KUKA KRL program: MyProgram_199().src

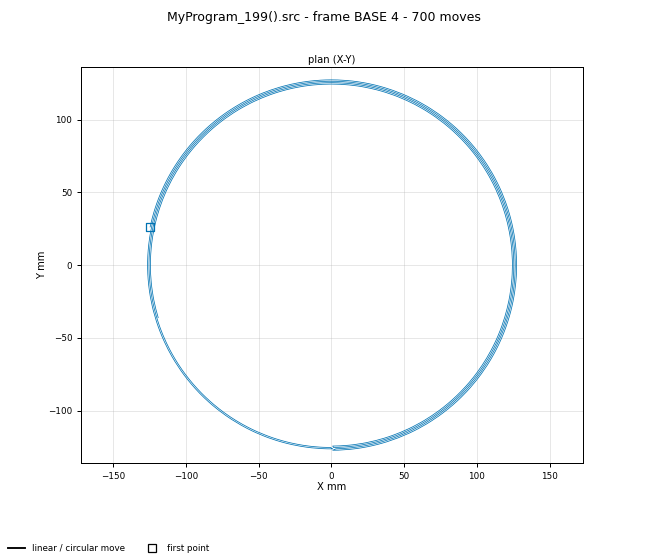
[picture p0: tool path of MyProgram_199().src in frame BASE 4, 700 of 700 moves have a stored position in this frame; points joined in program order, loops and branches not executed]
&ACCESS RVP
&REL 1
&PARAM TEMPLATE = C:\KRC\Roboter\Template\vorgabe
&PARAM EDITMASK = *
DEF MyProgram_199()
; ---- Setting reference (Base) ----
$BASE = BASE_DATA[4]

; --------------------------
; ---- Setting tool (TCP) ----
$TOOL = TOOL_DATA[3]
; --------------------------

$VEL.CP = VEL_APROX_PRINT
Startdeposition()
$VEL.CP = VEL_PRINT
LIN {X -124.5272,Y 26.175,Z 143,A 164.1665,B 24.1206,C -1.3898,E1 24.0018,E2 642.4936} C_DIS
LIN {X -123.2727,Y 31.5525,Z 143,A 161.827,B 24.1198,C -1.4042,E1 24.0033,E2 644.8119} C_DIS
LIN {X -122.0443,Y 36.0123,Z 143,A 159.352,B 24.1204,C -1.3939,E1 24.0052,E2 647.3273} C_DIS
LIN {X -120.9556,Y 39.5205,Z 143,A 158.1178,B 24.1191,C -1.4173,E1 24.0063,E2 648.5112} C_DIS
LIN {X -119.8977,Y 42.6203,Z 143,A 156.6922,B 24.1187,C -1.4241,E1 24.0075,E2 649.9285} C_DIS
LIN {X -118.7019,Y 45.8427,Z 143,A 154.9477,B 24.1189,C -1.4203,E1 24.0093,E2 651.6925} C_DIS
LIN {X -117.3172,Y 49.2782,Z 143,A 152.7105,B 24.12,C -1.4008,E1 24.0118,E2 653.9905} C_DIS
LIN {X -115.3752,Y 53.668,Z 143,A 151.1857,B 24.1181,C -1.435,E1 24.0135,E2 655.44} C_DIS
LIN {X -114.0458,Y 56.4373,Z 143,A 149.7836,B 24.1179,C -1.4383,E1 24.0152,E2 656.8417} C_DIS
LIN {X -112.4501,Y 59.5546,Z 143,A 147.9643,B 24.1183,C -1.4324,E1 24.0175,E2 658.6856} C_DIS
LIN {X -109.8769,Y 64.1814,Z 143,A 145.6973,B 24.1176,C -1.4445,E1 24.0207,E2 660.9353} C_DIS
LIN {X -107.6931,Y 67.7812,Z 143,A 143.7781,B 24.1173,C -1.4489,E1 24.0235,E2 662.8538} C_DIS
LIN {X -105.2252,Y 71.5528,Z 143,A 141.7365,B 24.1171,C -1.4541,E1 24.0266,E2 664.8932} C_DIS
LIN {X -102.675,Y 75.1662,Z 143,A 139.7684,B 24.1167,C -1.4606,E1 24.0298,E2 666.8553} C_DIS
LIN {X -100.2448,Y 78.3782,Z 143,A 137.8484,B 24.1167,C -1.4608,E1 24.0331,E2 668.7842} C_DIS
LIN {X -97.0311,Y 82.3229,Z 143,A 135.7966,B 24.1157,C -1.4774,E1 24.0367,E2 670.8052} C_DIS
LIN {X -94.8087,Y 84.8728,Z 143,A 133.5905,B 24.1172,C -1.4513,E1 24.0409,E2 673.0856} C_DIS
LIN {X -91.6928,Y 88.2304,Z 143,A 131.505,B 24.117,C -1.4554,E1 24.045,E2 675.1704} C_DIS
LIN {X -88.4466,Y 91.4838,Z 143,A 130.1435,B 24.1149,C -1.4916,E1 24.0475,E2 676.449} C_DIS
LIN {X -85.9693,Y 93.8157,Z 143,A 127.9481,B 24.1164,C -1.4659,E1 24.0522,E2 678.7167} C_DIS
LIN {X -82.7807,Y 96.64,Z 143,A 126.4601,B 24.115,C -1.4892,E1 24.0552,E2 680.1535} C_DIS
LIN {X -79.8951,Y 99.0396,Z 143,A 124.7629,B 24.1148,C -1.4926,E1 24.0589,E2 681.849} C_DIS
LIN {X -76.5158,Y 101.6731,Z 143,A 122.8099,B 24.1147,C -1.4957,E1 24.0632,E2 683.8019} C_DIS
LIN {X -72.9495,Y 104.2619,Z 143,A 120.7574,B 24.1147,C -1.4967,E1 24.0679,E2 685.8592} C_DIS
LIN {X -70.0309,Y 106.2438,Z 143,A 119.2441,B 24.1142,C -1.5032,E1 24.0714,E2 687.3619} C_DIS
LIN {X -66.2642,Y 108.6335,Z 143,A 116.7258,B 24.1153,C -1.4842,E1 24.0775,E2 689.9348} C_DIS
LIN {X -62.3439,Y 110.9293,Z 143,A 115.1658,B 24.1139,C -1.5095,E1 24.0811,E2 691.4375} C_DIS
LIN {X -58.8236,Y 112.834,Z 143,A 113.4971,B 24.1133,C -1.5186,E1 24.0852,E2 693.0888} C_DIS
LIN {X -56.2226,Y 114.1518,Z 143,A 112.1566,B 24.1133,C -1.5195,E1 24.0886,E2 694.4308} C_DIS
LIN {X -53.1753,Y 115.603,Z 143,A 110.5764,B 24.1133,C -1.5191,E1 24.0926,E2 696.016} C_DIS
LIN {X -50.3374,Y 116.8665,Z 143,A 109.2109,B 24.1131,C -1.5227,E1 24.096,E2 697.3761} C_DIS
LIN {X -47.1249,Y 118.1994,Z 143,A 106.7623,B 24.1153,C -1.4852,E1 24.1027,E2 699.9222} C_DIS
LIN {X -41.565,Y 120.2663,Z 143,A 104.0516,B 24.1152,C -1.4868,E1 24.1098,E2 702.6346} C_DIS
LIN {X -35.7294,Y 122.1272,Z 143,A 102.2253,B 24.1125,C -1.5319,E1 24.1144,E2 704.3534} C_DIS
LIN {X -32.6041,Y 122.9986,Z 143,A 100.6987,B 24.1126,C -1.5304,E1 24.1185,E2 705.8861} C_DIS
LIN {X -27.5686,Y 124.2263,Z 143,A 98.4289,B 24.1123,C -1.5355,E1 24.1247,E2 708.1466} C_DIS
LIN {X -23.6156,Y 125.0362,Z 143,A 96.5708,B 24.1123,C -1.5351,E1 24.1298,E2 710.0079} C_DIS
LIN {X -19.7127,Y 125.7106,Z 143,A 94.7472,B 24.1123,C -1.5346,E1 24.1348,E2 711.8346} C_DIS
LIN {X -16.2002,Y 126.2116,Z 143,A 93.0887,B 24.1125,C -1.5327,E1 24.1394,E2 713.4988} C_DIS
LIN {X -12.0343,Y 126.6763,Z 143,A 91.2754,B 24.1122,C -1.5372,E1 24.1444,E2 715.3025} C_DIS
LIN {X -7.2561,Y 127.0405,Z 143,A 88.7598,B 24.1131,C -1.5215,E1 24.1515,E2 717.8573} C_DIS
LIN {X -3.7963,Y 127.1904,Z 143,A 87.5723,B 24.1121,C -1.5392,E1 24.1547,E2 719.0017} C_DIS
LIN {X -0.1288,Y 127.248,Z 143,A 85.3654,B 24.1136,C -1.5137,E1 24.1611,E2 721.2708} C_DIS
LIN {X 4.2966,Y 127.1759,Z 143,A 83.9944,B 24.1119,C -1.5428,E1 24.1647,E2 722.5704} C_DIS
LIN {X 7.6952,Y 127.0138,Z 143,A 82.4885,B 24.1118,C -1.5441,E1 24.1689,E2 724.0726} C_DIS
LIN {X 10.3341,Y 126.8269,Z 143,A 81.1022,B 24.1123,C -1.5349,E1 24.1728,E2 725.4807} C_DIS
LIN {X 14.3391,Y 126.4382,Z 143,A 79.2362,B 24.1125,C -1.532,E1 24.178,E2 727.3524} C_DIS
LIN {X 18.3253,Y 125.9205,Z 143,A 77.4824,B 24.1124,C -1.5342,E1 24.1828,E2 729.0993} C_DIS
LIN {X 22.3665,Y 125.2654,Z 143,A 75.7321,B 24.1122,C -1.5379,E1 24.1876,E2 730.8386} C_DIS
LIN {X 25.9022,Y 124.5834,Z 143,A 73.9894,B 24.1126,C -1.5314,E1 24.1924,E2 732.595} C_DIS
LIN {X 29.705,Y 123.7307,Z 143,A 72.3528,B 24.1123,C -1.5361,E1 24.1969,E2 734.2179} C_DIS
LIN {X 32.889,Y 122.9226,Z 143,A 70.8777,B 24.1123,C -1.5353,E1 24.2008,E2 735.6924} C_DIS
LIN {X 36.7581,Y 121.8225,Z 143,A 68.3038,B 24.1145,C -1.4979,E1 24.208,E2 738.3531} C_DIS
LIN {X 41.983,Y 120.1214,Z 143,A 66.8144,B 24.1119,C -1.5425,E1 24.2116,E2 739.7305} C_DIS
LIN {X 48.6266,Y 117.5894,Z 143,A 63.5741,B 24.1122,C -1.5374,E1 24.2201,E2 742.976} C_DIS
LIN {X 52.3171,Y 115.9943,Z 143,A 61.5114,B 24.113,C -1.5232,E1 24.2254,E2 745.0681} C_DIS
LIN {X 57.8621,Y 113.3296,Z 143,A 58.8534,B 24.113,C -1.5251,E1 24.2321,E2 747.7141} C_DIS
LIN {X 60.9839,Y 111.6828,Z 143,A 57.1789,B 24.1133,C -1.5187,E1 24.2362,E2 749.3991} C_DIS
LIN {X 65.2332,Y 109.2553,Z 143,A 55.1366,B 24.113,C -1.5233,E1 24.2411,E2 751.4238} C_DIS
LIN {X 68.3421,Y 107.3384,Z 143,A 53.2984,B 24.1137,C -1.5113,E1 24.2455,E2 753.2852} C_DIS
LIN {X 73.4348,Y 103.9202,Z 143,A 50.8446,B 24.1131,C -1.5217,E1 24.2511,E2 755.7051} C_DIS
LIN {X 75.7493,Y 102.2458,Z 143,A 49.305,B 24.114,C -1.507,E1 24.2546,E2 757.2748} C_DIS
LIN {X 79.2546,Y 99.5529,Z 143,A 47.3269,B 24.1142,C -1.5039,E1 24.259,E2 759.2528} C_DIS
LIN {X 82.6863,Y 96.7222,Z 143,A 45.3026,B 24.1145,C -1.499,E1 24.2633,E2 761.281} C_DIS
LIN {X 85.935,Y 93.8473,Z 143,A 43.3542,B 24.1147,C -1.4953,E1 24.2673,E2 763.2304} C_DIS
LIN {X 89.2409,Y 90.7093,Z 143,A 41.3376,B 24.1148,C -1.4926,E1 24.2714,E2 765.2447} C_DIS
LIN {X 92.2645,Y 87.6327,Z 143,A 39.4106,B 24.115,C -1.4891,E1 24.2751,E2 767.1717} C_DIS
LIN {X 95.0993,Y 84.5477,Z 143,A 37.4842,B 24.1154,C -1.4828,E1 24.2788,E2 769.1045} C_DIS
LIN {X 98.0466,Y 81.1107,Z 143,A 35.1728,B 24.1165,C -1.4645,E1 24.283,E2 771.4495} C_DIS
LIN {X 100.4117,Y 78.1641,Z 143,A 34.1152,B 24.1149,C -1.4922,E1 24.2847,E2 772.4343} C_DIS
LIN {X 102.2377,Y 75.7602,Z 143,A 32.4351,B 24.116,C -1.4729,E1 24.2875,E2 774.1532} C_DIS
LIN {X 104.9494,Y 71.9562,Z 143,A 30.3694,B 24.1162,C -1.4694,E1 24.2909,E2 776.217} C_DIS
LIN {X 107.1146,Y 68.6917,Z 143,A 28.6075,B 24.1164,C -1.4649,E1 24.2935,E2 777.9808} C_DIS
LIN {X 110.4405,Y 63.2061,Z 143,A 26.0074,B 24.1161,C -1.4715,E1 24.2972,E2 780.5509} C_DIS
LIN {X 111.9201,Y 60.5483,Z 143,A 24.3472,B 24.1171,C -1.4531,E1 24.2995,E2 782.2467} C_DIS
LIN {X 114.1794,Y 56.1666,Z 143,A 22.2677,B 24.1171,C -1.4539,E1 24.3021,E2 784.3128} C_DIS
LIN {X 115.6591,Y 53.0539,Z 143,A 20.7526,B 24.1172,C -1.4513,E1 24.3039,E2 785.8258} C_DIS
LIN {X 116.9946,Y 50.0412,Z 143,A 18.1864,B 24.1204,C -1.393,E1 24.3069,E2 788.5191} C_DIS
LIN {X 119.5516,Y 43.5801,Z 143,A 15.4723,B 24.1198,C -1.4042,E1 24.3094,E2 791.1903} C_DIS
LIN {X 121.1576,Y 38.8909,Z 143,A 13.3661,B 24.1198,C -1.4037,E1 24.3112,E2 793.2853} C_DIS
LIN {X 122.4466,Y 34.6207,Z 143,A 12.1149,B 24.1181,C -1.4356,E1 24.3121,E2 794.4515} C_DIS
LIN {X 123.2167,Y 31.773,Z 143,A 10.5319,B 24.119,C -1.4186,E1 24.3133,E2 796.0665} C_DIS
LIN {X 124.0498,Y 28.3427,Z 143,A 8.9948,B 24.1192,C -1.4162,E1 24.3143,E2 797.6} C_DIS
LIN {X 124.7446,Y 25.1102,Z 143,A 7.5368,B 24.1193,C -1.4131,E1 24.3151,E2 799.0569} C_DIS
LIN {X 125.4856,Y 21.0966,Z 143,A 5.7162,B 24.1196,C -1.4081,E1 24.316,E2 800.8785} C_DIS
LIN {X 126.0104,Y 17.6965,Z 143,A 4.0643,B 24.1202,C -1.398,E1 24.3167,E2 802.5449} C_DIS
LIN {X 126.5349,Y 13.4408,Z 143,A 2.2564,B 24.1202,C -1.398,E1 24.3172,E2 804.3417} C_DIS
LIN {X 126.8936,Y 9.475,Z 143,A 0.4251,B 24.1206,C -1.3902,E1 24.3177,E2 806.1805} C_DIS
LIN {X 127.2222,Y 2.5341,Z 143,A -2.4521,B 24.1205,C -1.3928,E1 24.318,E2 809.0338} C_DIS
LIN {X 127.1851,Y -3.9522,Z 143,A -5.6524,B 24.1217,C -1.369,E1 24.318,E2 812.272} C_DIS
LIN {X 127.0034,Y -7.8649,Z 143,A -7.2947,B 24.1217,C -1.3694,E1 24.3177,E2 813.9033} C_DIS
LIN {X 126.673,Y -12.0688,Z 143,A -9.1796,B 24.122,C -1.3639,E1 24.3172,E2 815.79} C_DIS
LIN {X 125.9979,Y -17.7836,Z 143,A -11.5619,B 24.1219,C -1.366,E1 24.3164,E2 818.1524} C_DIS
LIN {X 125.5414,Y -20.7622,Z 143,A -13.1259,B 24.1227,C -1.3511,E1 24.3157,E2 819.7433} C_DIS
LIN {X 124.8202,Y -24.7388,Z 143,A -15.3256,B 24.124,C -1.3259,E1 24.3145,E2 821.9908} C_DIS
LIN {X 124.0308,Y -28.4258,Z 143,A -16.5022,B 24.1229,C -1.3468,E1 24.3138,E2 823.1094} C_DIS
LIN {X 123.3013,Y -31.4399,Z 143,A -17.9511,B 24.1233,C -1.3397,E1 24.3128,E2 824.5671} C_DIS
LIN {X 122.3396,Y -35.0032,Z 143,A -20.1035,B 24.1248,C -1.3095,E1 24.3112,E2 826.78} C_DIS
LIN {X 121.1722,Y -38.8452,Z 143,A -21.418,B 24.1239,C -1.3287,E1 24.3101,E2 828.0401} C_DIS
LIN {X 119.4922,Y -43.745,Z 143,A -23.6832,B 24.1241,C -1.3247,E1 24.308,E2 830.3016} C_DIS
LIN {X 118.3727,Y -46.6894,Z 143,A -25.5245,B 24.1254,C -1.2989,E1 24.3061,E2 832.1951} C_DIS
LIN {X 117.0359,Y -49.9411,Z 143,A -27.4139,B 24.1264,C -1.2787,E1 24.304,E2 834.1231} C_DIS
LIN {X 114.8725,Y -54.735,Z 143,A -28.7689,B 24.1242,C -1.3226,E1 24.3025,E2 835.3636} C_DIS
LIN {X 113.2953,Y -57.9294,Z 143,A -30.6449,B 24.1251,C -1.3039,E1 24.3001,E2 837.2746} C_DIS
LIN {X 111.5668,Y -61.1965,Z 143,A -32.3955,B 24.1256,C -1.2945,E1 24.2978,E2 839.0385} C_DIS
LIN {X 109.5112,Y -64.8038,Z 143,A -34.2914,B 24.1259,C -1.2877,E1 24.2951,E2 840.9408} C_DIS
LIN {X 106.9666,Y -68.9229,Z 143,A -37.4263,B 24.1286,C -1.2337,E1 24.2902,E2 844.1907} C_DIS
LIN {X 102.9212,Y -74.8288,Z 143,A -39.4667,B 24.1261,C -1.2838,E1 24.2871,E2 846.0989} C_DIS
LIN {X 99.7193,Y -79.045,Z 143,A -42.1819,B 24.1273,C -1.2607,E1 24.2824,E2 848.8571} C_DIS
LIN {X 95.2135,Y -84.4186,Z 143,A -44.9279,B 24.1267,C -1.273,E1 24.2775,E2 851.56} C_DIS
LIN {X 92.859,Y -87.0024,Z 143,A -46.6893,B 24.1273,C -1.2596,E1 24.2741,E2 853.346} C_DIS
LIN {X 88.9185,Y -91.0254,Z 143,A -49.4625,B 24.1282,C -1.2415,E1 24.2686,E2 856.1511} C_DIS
LIN {X 86.4722,Y -93.3528,Z 143,A -50.6453,B 24.1276,C -1.2547,E1 24.2663,E2 857.2968} C_DIS
LIN {X 83.4676,Y -96.0484,Z 143,A -52.5339,B 24.128,C -1.2469,E1 24.2623,E2 859.1965} C_DIS
LIN {X 79.6258,Y -99.2568,Z 143,A -55.2366,B 24.1293,C -1.2196,E1 24.2563,E2 861.9551} C_DIS
LIN {X 76.152,Y -101.946,Z 143,A -56.4363,B 24.1276,C -1.254,E1 24.2539,E2 863.0665} C_DIS
LIN {X 73.7292,Y -103.7121,Z 143,A -58.3085,B 24.129,C -1.2252,E1 24.2495,E2 865.0021} C_DIS
LIN {X 68.4798,Y -107.2502,Z 143,A -60.5853,B 24.1279,C -1.248,E1 24.2443,E2 867.2154} C_DIS
LIN {X 65.0588,Y -109.3592,Z 143,A -62.7183,B 24.1289,C -1.2285,E1 24.2391,E2 869.3889} C_DIS
LIN {X 59.4478,Y -112.5062,Z 143,A -65.3808,B 24.1285,C -1.2349,E1 24.2327,E2 872.0277} C_DIS
LIN {X 57.032,Y -113.7522,Z 143,A -66.8895,B 24.1293,C -1.2188,E1 24.2288,E2 873.5714} C_DIS
LIN {X 53.4352,Y -115.4828,Z 143,A -68.5743,B 24.1292,C -1.2215,E1 24.2246,E2 875.2452} C_DIS
LIN {X 45.816,Y -118.7123,Z 143,A -71.9325,B 24.1286,C -1.2341,E1 24.2161,E2 878.5644} C_DIS
LIN {X 38.1325,Y -121.3998,Z 143,A -75.7888,B 24.1293,C -1.2198,E1 24.2059,E2 882.4475} C_DIS
LIN {X 34.5937,Y -122.4542,Z 143,A -77.3703,B 24.1292,C -1.2219,E1 24.2016,E2 884.021} C_DIS
LIN {X 31.4599,Y -123.2962,Z 143,A -79.0235,B 24.1297,C -1.211,E1 24.1971,E2 885.6982} C_DIS
LIN {X 28.2059,Y -124.081,Z 143,A -80.5262,B 24.1297,C -1.2098,E1 24.193,E2 887.2017} C_DIS
LIN {X 24.8866,Y -124.7901,Z 143,A -82.181,B 24.1301,C -1.2023,E1 24.1884,E2 888.8727} C_DIS
LIN {X 20.9689,Y -125.5069,Z 143,A -83.8399,B 24.1299,C -1.2074,E1 24.1839,E2 890.5173} C_DIS
LIN {X 17.5219,Y -126.0353,Z 143,A -85.6002,B 24.1303,C -1.1971,E1 24.179,E2 892.3011} C_DIS
LIN {X 12.5269,Y -126.6291,Z 143,A -87.4842,B 24.1295,C -1.2142,E1 24.1739,E2 894.142} C_DIS
LIN {X 4.6976,Y -127.1602,Z 143,A -91.0863,B 24.1298,C -1.2093,E1 24.1638,E2 897.7545} C_DIS
LIN {X 0.9052,Y -127.2215,Z 143,A -92.4328,B 24.1289,C -1.2265,E1 24.1602,E2 899.0586} C_DIS
Enddeposition()
LIN {X 0.9052,Y -127.2215,Z 143,A -92.4328,B 24.1289,C -1.2265,E1 24.1602,E2 899.0586} C_DIS
Startdeposition()
$VEL.CP = VEL_PRINT
LIN {X 3.0703,Y -126.2444,Z 143,A -90.8348,B 23.3783,C -1.1238,E1 23.4098,E2 897.6156} C_DIS
LIN {X 9.0133,Y -125.959,Z 143,A -88.2436,B 23.3785,C -1.1199,E1 23.4169,E2 895.0355} C_DIS
LIN {X 12.8377,Y -125.6284,Z 143,A -86.5864,B 23.3786,C -1.1168,E1 23.4215,E2 893.3871} C_DIS
LIN {X 17.843,Y -125.0139,Z 143,A -84.275,B 23.3786,C -1.1194,E1 23.4279,E2 891.0714} C_DIS
LIN {X 21.7376,Y -124.3968,Z 143,A -82.4343,B 23.3784,C -1.1231,E1 23.433,E2 889.2232} C_DIS
LIN {X 25.0313,Y -123.7751,Z 143,A -80.9906,B 23.3784,C -1.1208,E1 23.437,E2 887.7872} C_DIS
LIN {X 28.5169,Y -123.0193,Z 143,A -79.268,B 23.3782,C -1.1272,E1 23.4417,E2 886.051} C_DIS
LIN {X 32.3455,Y -122.068,Z 143,A -77.6252,B 23.3784,C -1.1221,E1 23.4461,E2 884.4238} C_DIS
LIN {X 35.6782,Y -121.1359,Z 143,A -75.87,B 23.3779,C -1.1326,E1 23.4509,E2 882.6453} C_DIS
LIN {X 42.4632,Y -118.9277,Z 143,A -72.6202,B 23.3777,C -1.1372,E1 23.4595,E2 879.3908} C_DIS
LIN {X 46.97,Y -117.2205,Z 143,A -70.8654,B 23.3785,C -1.1196,E1 23.4639,E2 877.6844} C_DIS
LIN {X 52.3569,Y -114.9174,Z 143,A -67.8848,B 23.3776,C -1.1389,E1 23.4717,E2 874.6631} C_DIS
LIN {X 55.7551,Y -113.3055,Z 143,A -66.2507,B 23.3776,C -1.1382,E1 23.4757,E2 873.0354} C_DIS
LIN {X 61.2211,Y -110.45,Z 143,A -63.4821,B 23.3776,C -1.1415,E1 23.4826,E2 870.2669} C_DIS
LIN {X 64.3168,Y -108.6772,Z 143,A -61.8595,B 23.3774,C -1.1446,E1 23.4865,E2 868.6418} C_DIS
LIN {X 67.2956,Y -106.8576,Z 143,A -60.2613,B 23.3772,C -1.1483,E1 23.4903,E2 867.0397} C_DIS
LIN {X 69.4871,Y -105.4456,Z 143,A -59.0358,B 23.377,C -1.1527,E1 23.4932,E2 865.8076} C_DIS
LIN {X 74.8729,Y -101.6922,Z 143,A -56.0676,B 23.3767,C -1.1583,E1 23.4999,E2 862.8364} C_DIS
LIN {X 78.5319,Y -98.8938,Z 143,A -53.9887,B 23.3766,C -1.1623,E1 23.5045,E2 860.7558} C_DIS
LIN {X 83.5514,Y -94.6911,Z 143,A -51.0321,B 23.3763,C -1.1683,E1 23.5108,E2 857.7965} C_DIS
LIN {X 88.903,Y -89.6855,Z 143,A -47.0482,B 23.3743,C -1.2087,E1 23.519,E2 853.7291} C_DIS
LIN {X 92.7346,Y -85.7184,Z 143,A -45.2748,B 23.3758,C -1.179,E1 23.5222,E2 852.0384} C_DIS
LIN {X 97.8322,Y -79.8504,Z 143,A -40.9889,B 23.3735,C -1.2257,E1 23.5301,E2 847.6566} C_DIS
LIN {X 101.4084,Y -75.257,Z 143,A -39.1077,B 23.375,C -1.1953,E1 23.5331,E2 845.8614} C_DIS
LIN {X 103.0955,Y -72.9286,Z 143,A -36.7932,B 23.3723,C -1.249,E1 23.537,E2 843.4244} C_DIS
LIN {X 107.074,Y -66.9512,Z 143,A -34.5488,B 23.3744,C -1.2078,E1 23.5402,E2 841.2955} C_DIS
LIN {X 109.3173,Y -63.2216,Z 143,A -32.6201,B 23.3742,C -1.2113,E1 23.5429,E2 839.3688} C_DIS
LIN {X 111.3593,Y -59.5517,Z 143,A -30.6871,B 23.3739,C -1.2182,E1 23.5455,E2 837.4292} C_DIS
LIN {X 113.161,Y -56.048,Z 143,A -29.16,B 23.3742,C -1.2108,E1 23.5474,E2 835.9295} C_DIS
LIN {X 116.3932,Y -48.9847,Z 143,A -25.5078,B 23.3734,C -1.2277,E1 23.5516,E2 832.2563} C_DIS
LIN {X 117.5948,Y -46.0252,Z 143,A -24.1792,B 23.3734,C -1.2262,E1 23.553,E2 830.9393} C_DIS
LIN {X 118.592,Y -43.3943,Z 143,A -22.4227,B 23.3721,C -1.2539,E1 23.5547,E2 829.1239} C_DIS
LIN {X 119.7735,Y -40.0138,Z 143,A -21.3647,B 23.3732,C -1.231,E1 23.5556,E2 828.13} C_DIS
LIN {X 121.5558,Y -34.2204,Z 143,A -18.5087,B 23.3725,C -1.2448,E1 23.5579,E2 825.2567} C_DIS
LIN {X 122.3741,Y -31.1673,Z 143,A -17.1035,B 23.3724,C -1.248,E1 23.5589,E2 823.8523} C_DIS
LIN {X 123.4702,Y -26.4942,Z 143,A -14.8735,B 23.3719,C -1.2575,E1 23.5603,E2 821.6123} C_DIS
LIN {X 124.2579,Y -22.5139,Z 143,A -13.0509,B 23.3716,C -1.2625,E1 23.5613,E2 819.7887} C_DIS
LIN {X 124.864,Y -18.8685,Z 143,A -10.8775,B 23.3701,C -1.2926,E1 23.5622,E2 817.5537} C_DIS
LIN {X 125.4288,Y -14.6483,Z 143,A -9.4064,B 23.371,C -1.276,E1 23.5627,E2 816.1336} C_DIS
LIN {X 125.8412,Y -10.5292,Z 143,A -7.6065,B 23.3708,C -1.2782,E1 23.5631,E2 814.3396} C_DIS
LIN {X 126.0963,Y -6.8457,Z 143,A -6.0912,B 23.371,C -1.2757,E1 23.5634,E2 812.8403} C_DIS
LIN {X 126.2797,Y -0.8325,Z 143,A -3.6263,B 23.3712,C -1.2715,E1 23.5636,E2 810.4018} C_DIS
LIN {X 126.2604,Y 2.2898,Z 143,A -1.8926,B 23.3701,C -1.2917,E1 23.5636,E2 808.6286} C_DIS
LIN {X 126.0769,Y 7.1985,Z 143,A 0.3117,B 23.3698,C -1.2976,E1 23.5633,E2 806.4235} C_DIS
LIN {X 125.8526,Y 10.3945,Z 143,A 1.8479,B 23.3694,C -1.3064,E1 23.563,E2 804.8751} C_DIS
LIN {X 125.4982,Y 14.048,Z 143,A 3.5727,B 23.3689,C -1.3146,E1 23.5624,E2 803.1407} C_DIS
LIN {X 125.0207,Y 17.7952,Z 143,A 5.1722,B 23.3689,C -1.3145,E1 23.5619,E2 801.5518} C_DIS
LIN {X 124.4344,Y 21.5277,Z 143,A 6.8886,B 23.3686,C -1.32,E1 23.5611,E2 799.8324} C_DIS
LIN {X 123.7908,Y 24.954,Z 143,A 8.4425,B 23.3685,C -1.3236,E1 23.5602,E2 798.2792} C_DIS
LIN {X 123.0633,Y 28.3247,Z 143,A 10.0144,B 23.3682,C -1.3288,E1 23.5593,E2 796.704} C_DIS
LIN {X 122.0814,Y 32.2955,Z 143,A 11.7987,B 23.3681,C -1.331,E1 23.5581,E2 794.9253} C_DIS
LIN {X 121.1474,Y 35.6388,Z 143,A 14.0642,B 23.3659,C -1.37,E1 23.5562,E2 792.5762} C_DIS
LIN {X 119.6438,Y 40.4033,Z 143,A 15.7815,B 23.3671,C -1.3496,E1 23.5548,E2 790.9204} C_DIS
LIN {X 118.3757,Y 43.9782,Z 143,A 17.2604,B 23.3674,C -1.3429,E1 23.5534,E2 789.4673} C_DIS
LIN {X 116.1309,Y 49.6053,Z 143,A 20.1647,B 23.3666,C -1.3585,E1 23.5503,E2 786.5411} C_DIS
LIN {X 114.8576,Y 52.4863,Z 143,A 21.6205,B 23.3663,C -1.3639,E1 23.5486,E2 785.0803} C_DIS
LIN {X 112.9208,Y 56.5349,Z 143,A 23.7059,B 23.3658,C -1.372,E1 23.546,E2 782.9865} C_DIS
LIN {X 110.8846,Y 60.4304,Z 143,A 25.2832,B 23.3666,C -1.3572,E1 23.544,E2 781.4553} C_DIS
LIN {X 109.4448,Y 62.9996,Z 143,A 27.2771,B 23.3647,C -1.3929,E1 23.5412,E2 779.3829} C_DIS
LIN {X 107.4784,Y 66.3002,Z 143,A 28.669,B 23.3654,C -1.3804,E1 23.5392,E2 778.0301} C_DIS
LIN {X 105.2267,Y 69.819,Z 143,A 30.5814,B 23.365,C -1.3861,E1 23.5363,E2 776.1136} C_DIS
LIN {X 102.9014,Y 73.2022,Z 143,A 32.4389,B 23.3648,C -1.3906,E1 23.5333,E2 774.2546} C_DIS
LIN {X 100.3238,Y 76.6966,Z 143,A 34.5444,B 23.3641,C -1.4021,E1 23.5297,E2 772.1312} C_DIS
LIN {X 96.7287,Y 81.1836,Z 143,A 36.9626,B 23.3643,C -1.3991,E1 23.5255,E2 769.7326} C_DIS
LIN {X 93.8377,Y 84.5094,Z 143,A 38.9811,B 23.364,C -1.4046,E1 23.5217,E2 767.7101} C_DIS
LIN {X 90.8868,Y 87.6748,Z 143,A 40.9026,B 23.3639,C -1.4069,E1 23.518,E2 765.7917} C_DIS
LIN {X 87.9767,Y 90.5945,Z 143,A 42.7877,B 23.3636,C -1.4116,E1 23.5143,E2 763.9033} C_DIS
LIN {X 84.6059,Y 93.7506,Z 143,A 44.8759,B 23.3634,C -1.4156,E1 23.51,E2 761.8142} C_DIS
LIN {X 81.3687,Y 96.5734,Z 143,A 46.8072,B 23.3632,C -1.4186,E1 23.5059,E2 759.8836} C_DIS
LIN {X 78.0166,Y 99.3007,Z 143,A 48.5897,B 23.3635,C -1.4138,E1 23.502,E2 758.1204} C_DIS
LIN {X 75.0876,Y 101.5344,Z 143,A 50.2862,B 23.3632,C -1.418,E1 23.4983,E2 756.4199} C_DIS
LIN {X 71.4837,Y 104.1022,Z 143,A 52.5264,B 23.3624,C -1.4324,E1 23.4931,E2 754.1517} C_DIS
LIN {X 67.4019,Y 106.7905,Z 143,A 54.5602,B 23.3627,C -1.4273,E1 23.4883,E2 752.138} C_DIS
LIN {X 64.1824,Y 108.7562,Z 143,A 56.0506,B 23.3631,C -1.4194,E1 23.4848,E2 750.6723} C_DIS
LIN {X 61.8868,Y 110.0784,Z 143,A 57.5822,B 23.3621,C -1.4367,E1 23.481,E2 749.1022} C_DIS
LIN {X 58.555,Y 111.8843,Z 143,A 59.2144,B 23.3622,C -1.4349,E1 23.477,E2 747.4794} C_DIS
LIN {X 53.7161,Y 114.2889,Z 143,A 61.7393,B 23.3619,C -1.4414,E1 23.4707,E2 744.9454} C_DIS
LIN {X 50.168,Y 115.8876,Z 143,A 63.373,B 23.3621,C -1.4373,E1 23.4665,E2 743.3265} C_DIS
LIN {X 46.8946,Y 117.2509,Z 143,A 65.5891,B 23.3603,C -1.4674,E1 23.4606,E2 741.0399} C_DIS
LIN {X 42.404,Y 118.9491,Z 143,A 67.248,B 23.3617,C -1.4451,E1 23.4564,E2 739.4409} C_DIS
LIN {X 39.0441,Y 120.0948,Z 143,A 69.1038,B 23.3609,C -1.4578,E1 23.4514,E2 737.5567} C_DIS
LIN {X 35.8172,Y 121.0952,Z 143,A 70.2942,B 23.3618,C -1.4431,E1 23.4483,E2 736.4058} C_DIS
LIN {X 32.6406,Y 121.9893,Z 143,A 71.7276,B 23.3618,C -1.4411,E1 23.4445,E2 734.9798} C_DIS
LIN {X 29.5465,Y 122.7754,Z 143,A 73.2271,B 23.3618,C -1.4444,E1 23.4404,E2 733.4745} C_DIS
LIN {X 25.6496,Y 123.6493,Z 143,A 75.0835,B 23.3615,C -1.4473,E1 23.4353,E2 731.6132} C_DIS
LIN {X 21.7187,Y 124.4002,Z 143,A 76.8644,B 23.3615,C -1.4464,E1 23.4304,E2 729.8367} C_DIS
LIN {X 17.8497,Y 125.0129,Z 143,A 78.6606,B 23.3615,C -1.4479,E1 23.4255,E2 728.0388} C_DIS
LIN {X 13.7932,Y 125.5256,Z 143,A 80.4772,B 23.3615,C -1.4465,E1 23.4204,E2 726.2271} C_DIS
LIN {X 10.3945,Y 125.8526,Z 143,A 82.0898,B 23.3614,C -1.4495,E1 23.4159,E2 724.6078} C_DIS
LIN {X 7.597,Y 126.0523,Z 143,A 83.4759,B 23.3611,C -1.4547,E1 23.412,E2 723.2092} C_DIS
LIN {X 3.3796,Y 126.2358,Z 143,A 85.4736,B 23.3609,C -1.4583,E1 23.4064,E2 721.2029} C_DIS
LIN {X -1.4286,Y 126.2747,Z 143,A 87.4404,B 23.3615,C -1.4481,E1 23.401,E2 719.2619} C_DIS
LIN {X -4.5585,Y 126.1992,Z 143,A 88.7783,B 23.3617,C -1.444,E1 23.3973,E2 717.9342} C_DIS
LIN {X -10.2698,Y 125.8631,Z 143,A 91.4685,B 23.3615,C -1.4472,E1 23.3898,E2 715.2348} C_DIS
LIN {X -13.8004,Y 125.5248,Z 143,A 93.0275,B 23.3617,C -1.4442,E1 23.3855,E2 713.6827} C_DIS
LIN {X -17.827,Y 125.0162,Z 143,A 94.8643,B 23.3617,C -1.4428,E1 23.3804,E2 711.8477} C_DIS
LIN {X -21.5271,Y 124.4345,Z 143,A 96.6906,B 23.3615,C -1.4473,E1 23.3753,E2 710.0084} C_DIS
LIN {X -25.061,Y 123.7691,Z 143,A 98.1808,B 23.362,C -1.4397,E1 23.3713,E2 708.5355} C_DIS
LIN {X -28.2376,Y 123.0832,Z 143,A 99.7743,B 23.3617,C -1.4437,E1 23.3669,E2 706.9297} C_DIS
LIN {X -33.339,Y 121.8023,Z 143,A 102.1269,B 23.362,C -1.4398,E1 23.3606,E2 704.5832} C_DIS
LIN {X -37.8031,Y 120.4897,Z 143,A 104.6963,B 23.3609,C -1.4578,E1 23.3536,E2 701.9634} C_DIS
LIN {X -41.8081,Y 119.1599,Z 143,A 105.9845,B 23.3627,C -1.4277,E1 23.3504,E2 700.7487} C_DIS
LIN {X -46.4132,Y 117.4439,Z 143,A 108.3333,B 23.3625,C -1.43,E1 23.3442,E2 698.3889} C_DIS
LIN {X -49.7738,Y 116.058,Z 143,A 109.9891,B 23.3627,C -1.4279,E1 23.34,E2 696.7341} C_DIS
LIN {X -52.7954,Y 114.7147,Z 143,A 111.5069,B 23.3627,C -1.4265,E1 23.3361,E2 695.2161} C_DIS
LIN {X -55.7129,Y 113.3263,Z 143,A 112.9483,B 23.3629,C -1.4231,E1 23.3325,E2 693.7792} C_DIS
LIN {X -58.5976,Y 111.8619,Z 143,A 114.4346,B 23.363,C -1.4215,E1 23.3288,E2 692.2926} C_DIS
LIN {X -64.3759,Y 108.6415,Z 143,A 117.5772,B 23.363,C -1.4223,E1 23.3212,E2 689.138} C_DIS
LIN {X -68.2831,Y 106.2295,Z 143,A 119.6539,B 23.3632,C -1.4181,E1 23.3162,E2 687.0648} C_DIS
LIN {X -72.254,Y 103.5693,Z 143,A 121.8164,B 23.3635,C -1.4136,E1 23.3113,E2 684.906} C_DIS
LIN {X -75.7598,Y 101.0338,Z 143,A 123.8365,B 23.3635,C -1.412,E1 23.3067,E2 682.8822} C_DIS
LIN {X -79.2371,Y 98.3296,Z 143,A 125.7181,B 23.3641,C -1.4026,E1 23.3026,E2 681.0167} C_DIS
LIN {X -84.4846,Y 93.8598,Z 143,A 128.9271,B 23.3643,C -1.3991,E1 23.2959,E2 677.8032} C_DIS
LIN {X -87.4018,Y 91.1493,Z 143,A 130.7114,B 23.3646,C -1.3938,E1 23.2922,E2 676.0243} C_DIS
LIN {X -89.3186,Y 89.2723,Z 143,A 132.2048,B 23.3641,C -1.4028,E1 23.2892,E2 674.5014} C_DIS
LIN {X -93.7506,Y 84.606,Z 143,A 134.9303,B 23.365,C -1.3871,E1 23.2841,E2 671.8027} C_DIS
LIN {X -96.4924,Y 81.4651,Z 143,A 136.7123,B 23.3655,C -1.3776,E1 23.2809,E2 670.0362} C_DIS
LIN {X -99.6329,Y 77.5925,Z 143,A 139.1359,B 23.3655,C -1.3785,E1 23.2766,E2 667.5981} C_DIS
LIN {X -102.3893,Y 73.917,Z 143,A 141.1811,B 23.3659,C -1.3712,E1 23.2733,E2 665.5607} C_DIS
LIN {X -104.8565,Y 70.3736,Z 143,A 143.2061,B 23.366,C -1.3685,E1 23.2701,E2 663.5316} C_DIS
LIN {X -107.3404,Y 66.5231,Z 143,A 145.2673,B 23.3664,C -1.3619,E1 23.267,E2 661.4759} C_DIS
LIN {X -109.3173,Y 63.2216,Z 143,A 147.8961,B 23.3645,C -1.3947,E1 23.2632,E2 658.7491} C_DIS
LIN {X -112.354,Y 57.6496,Z 143,A 149.9142,B 23.3671,C -1.3493,E1 23.2607,E2 656.8347} C_DIS
LIN {X -113.7968,Y 54.7462,Z 143,A 152.1861,B 23.3654,C -1.3791,E1 23.2579,E2 654.4738} C_DIS
LIN {X -116.2741,Y 49.2698,Z 143,A 154.1725,B 23.3676,C -1.3391,E1 23.2558,E2 652.5772} C_DIS
LIN {X -117.64,Y 45.9089,Z 143,A 155.7794,B 23.368,C -1.3324,E1 23.2541,E2 650.9775} C_DIS
LIN {X -118.7982,Y 42.8224,Z 143,A 157.3054,B 23.3682,C -1.329,E1 23.2527,E2 649.4507} C_DIS
LIN {X -120.0208,Y 39.2711,Z 143,A 159.4798,B 23.3674,C -1.3437,E1 23.2507,E2 647.2258} C_DIS
LIN {X -121.2731,Y 35.2096,Z 143,A 160.9409,B 23.3688,C -1.3177,E1 23.2496,E2 645.8214} C_DIS
LIN {X -122.3497,Y 31.2634,Z 143,A 162.7802,B 23.3691,C -1.3111,E1 23.2483,E2 643.9872} C_DIS
LIN {X -123.2636,Y 27.4476,Z 143,A 164.8207,B 23.3688,C -1.3164,E1 23.247,E2 641.9204} C_DIS
LIN {X -124.2825,Y 22.3763,Z 143,A 166.9243,B 23.3698,C -1.2986,E1 23.2459,E2 639.8486} C_DIS
LIN {X -124.8786,Y 18.7743,Z 143,A 168.7514,B 23.3697,C -1.3005,E1 23.2451,E2 638.0051} C_DIS
LIN {X -125.4703,Y 14.3,Z 143,A 170.7671,B 23.3701,C -1.2925,E1 23.2445,E2 635.9967} C_DIS
LIN {X -125.8489,Y 10.4385,Z 143,A 172.4782,B 23.3705,C -1.2847,E1 23.244,E2 634.2941} C_DIS
LIN {X -126.1122,Y 6.5285,Z 143,A 174.2214,B 23.3709,C -1.2775,E1 23.2438,E2 632.558} C_DIS
LIN {X -126.2544,Y 2.6515,Z 143,A 176.0718,B 23.3709,C -1.2756,E1 23.2436,E2 630.7004} C_DIS
LIN {X -126.2656,Y -1.9732,Z 143,A 178.1088,B 23.3715,C -1.2662,E1 23.2436,E2 628.6739} C_DIS
LIN {X -126.136,Y -6.0547,Z 143,A 179.9925,B 23.3717,C -1.2616,E1 23.2438,E2 626.7898} C_DIS
LIN {X -125.8995,Y -9.8278,Z 143,A -178.2206,B 23.3718,C -1.2591,E1 23.2442,E2 624.9977} C_DIS
LIN {X -125.5539,Y -13.5299,Z 143,A -176.6044,B 23.3722,C -1.2507,E1 23.2447,E2 623.3922} C_DIS
LIN {X -125.0627,Y -17.5015,Z 143,A -174.7437,B 23.3724,C -1.2468,E1 23.2453,E2 621.5293} C_DIS
LIN {X -124.403,Y -21.7033,Z 143,A -172.7627,B 23.3726,C -1.2429,E1 23.2462,E2 619.5456} C_DIS
LIN {X -122.9701,Y -28.7314,Z 143,A -169.459,B 23.373,C -1.2348,E1 23.2482,E2 616.2415} C_DIS
LIN {X -122.3008,Y -31.4558,Z 143,A -167.0583,B 23.3708,C -1.2795,E1 23.2501,E2 613.7125} C_DIS
LIN {X -120.1658,Y -38.8218,Z 143,A -164.6405,B 23.3736,C -1.223,E1 23.2519,E2 611.4228} C_DIS
LIN {X -118.9169,Y -42.4932,Z 143,A -162.9365,B 23.374,C -1.2154,E1 23.2534,E2 609.7278} C_DIS
LIN {X -117.6484,Y -45.8873,Z 143,A -161.3145,B 23.3743,C -1.2096,E1 23.2551,E2 608.1105} C_DIS
LIN {X -116.0279,Y -49.8435,Z 143,A -159.4611,B 23.3747,C -1.2003,E1 23.257,E2 606.2698} C_DIS
LIN {X -114.713,Y -52.7989,Z 143,A -157.6592,B 23.3742,C -1.2104,E1 23.2592,E2 604.4314} C_DIS
LIN {X -112.1028,Y -58.1388,Z 143,A -155.0897,B 23.3749,C -1.1974,E1 23.2624,E2 601.8802} C_DIS
LIN {X -109.7588,Y -62.4521,Z 143,A -152.8697,B 23.3752,C -1.191,E1 23.2654,E2 599.6638} C_DIS
LIN {X -107.495,Y -66.2731,Z 143,A -150.8293,B 23.3754,C -1.1867,E1 23.2683,E2 597.623} C_DIS
LIN {X -103.5646,Y -72.2608,Z 143,A -147.6158,B 23.3759,C -1.1768,E1 23.2733,E2 594.4174} C_DIS
LIN {X -101.1887,Y -75.5519,Z 143,A -145.3789,B 23.3753,C -1.1894,E1 23.2771,E2 592.1368} C_DIS
LIN {X -98.8516,Y -78.5849,Z 143,A -143.996,B 23.3762,C -1.1698,E1 23.2794,E2 590.7967} C_DIS
LIN {X -96.1015,Y -81.9253,Z 143,A -142.0157,B 23.3764,C -1.1659,E1 23.283,E2 588.8164} C_DIS
LIN {X -93.2362,Y -85.1727,Z 143,A -140.0142,B 23.3765,C -1.163,E1 23.2867,E2 586.8126} C_DIS
LIN {X -90.3925,Y -88.1846,Z 143,A -138.1034,B 23.3766,C -1.1603,E1 23.2904,E2 584.8997} C_DIS
LIN {X -87.1702,Y -91.3706,Z 143,A -136.0982,B 23.377,C -1.1538,E1 23.2944,E2 582.9021} C_DIS
LIN {X -83.9952,Y -94.2982,Z 143,A -134.0888,B 23.377,C -1.152,E1 23.2986,E2 580.8885} C_DIS
LIN {X -81.5253,Y -96.4415,Z 143,A -131.9543,B 23.3758,C -1.178,E1 23.3033,E2 578.6793} C_DIS
LIN {X -77.358,Y -99.8146,Z 143,A -130.6121,B 23.3783,C -1.1252,E1 23.306,E2 577.4653} C_DIS
LIN {X -72.2892,Y -103.5448,Z 143,A -127.2922,B 23.3776,C -1.1407,E1 23.3136,E2 574.0937} C_DIS
LIN {X -68.487,Y -106.0984,Z 143,A -125.2483,B 23.3778,C -1.1358,E1 23.3183,E2 572.0549} C_DIS
LIN {X -61.918,Y -110.0608,Z 143,A -121.2516,B 23.3769,C -1.1539,E1 23.3281,E2 567.9997} C_DIS
LIN {X -57.9627,Y -112.1946,Z 143,A -119.6634,B 23.378,C -1.1309,E1 23.3319,E2 566.4648} C_DIS
LIN {X -54.6973,Y -113.8202,Z 143,A -118.0969,B 23.3783,C -1.1249,E1 23.3358,E2 564.909} C_DIS
LIN {X -51.7568,Y -115.1869,Z 143,A -116.6294,B 23.3783,C -1.1231,E1 23.3395,E2 563.4423} C_DIS
LIN {X -45.7981,Y -117.683,Z 143,A -113.7353,B 23.3786,C -1.1183,E1 23.347,E2 560.5531} C_DIS
LIN {X -43.1313,Y -118.6868,Z 143,A -112.5682,B 23.3789,C -1.1115,E1 23.35,E2 559.4008} C_DIS
LIN {X -37.967,Y -120.4389,Z 143,A -109.8631,B 23.3785,C -1.1199,E1 23.3572,E2 556.6692} C_DIS
LIN {X -34.2098,Y -121.5587,Z 143,A -108.14,B 23.3787,C -1.1161,E1 23.3618,E2 554.9525} C_DIS
LIN {X -30.9589,Y -122.427,Z 143,A -106.5892,B 23.3787,C -1.1163,E1 23.366,E2 553.3987} C_DIS
LIN {X -26.9283,Y -123.3765,Z 143,A -104.7474,B 23.3787,C -1.1136,E1 23.371,E2 551.5611} C_DIS
LIN {X -24.1141,Y -123.9577,Z 143,A -103.3968,B 23.3787,C -1.1152,E1 23.3748,E2 550.2048} C_DIS
LIN {X -21.2288,Y -124.4844,Z 143,A -101.5974,B 23.3778,C -1.1364,E1 23.3799,E2 548.3502} C_DIS
LIN {X -17.0657,Y -125.1241,Z 143,A -100.1242,B 23.3787,C -1.1157,E1 23.3838,E2 546.928} C_DIS
LIN {X -13.6189,Y -125.5444,Z 143,A -98.5973,B 23.3788,C -1.1132,E1 23.388,E2 545.4062} C_DIS
LIN {X -9.0536,Y -125.956,Z 143,A -96.5702,B 23.3789,C -1.1107,E1 23.3936,E2 543.3845} C_DIS
LIN {X -6.6834,Y -126.1044,Z 143,A -95.046,B 23.378,C -1.1315,E1 23.398,E2 541.8075} C_DIS
LIN {X -2.9369,Y -126.2481,Z 143,A -93.6317,B 23.3786,C -1.1183,E1 23.4019,E2 540.4262} C_DIS
LIN {X 0.9045,Y -126.2774,Z 143,A -92.6874,B 23.3802,C -1.0818,E1 23.4043,E2 539.5739} C_DIS
Enddeposition()
LIN {X 0.9045,Y -126.2774,Z 143,A -92.6874,B 23.3802,C -1.0818,E1 23.4043,E2 539.5739} C_DIS
Startdeposition()
$VEL.CP = VEL_PRINT
LIN {X -0.6601,Y -125.3135,Z 143,A -93.2281,B 22.5626,C -0.9537,E1 22.58,E2 540.3396} C_DIS
LIN {X -5.5186,Y -125.1952,Z 143,A -95.3408,B 22.5624,C -0.9582,E1 22.5741,E2 542.4409} C_DIS
LIN {X -8.1458,Y -125.0509,Z 143,A -96.7604,B 22.5628,C -0.9488,E1 22.5701,E2 543.8856} C_DIS
LIN {X -11.8994,Y -124.7489,Z 143,A -98.369,B 22.5626,C -0.9538,E1 22.5657,E2 545.4819} C_DIS
LIN {X -15.1247,Y -124.3993,Z 143,A -99.8439,B 22.5626,C -0.9544,E1 22.5616,E2 546.9564} C_DIS
LIN {X -19.6353,Y -123.768,Z 143,A -101.8601,B 22.5624,C -0.9578,E1 22.556,E2 548.9655} C_DIS
LIN {X -23.5142,Y -123.0891,Z 143,A -103.8032,B 22.5627,C -0.9524,E1 22.5506,E2 550.9251} C_DIS
LIN {X -27.7041,Y -122.2144,Z 143,A -105.6884,B 22.5625,C -0.9564,E1 22.5455,E2 552.8026} C_DIS
LIN {X -30.9677,Y -121.4284,Z 143,A -107.1471,B 22.5623,C -0.9605,E1 22.5416,E2 554.2527} C_DIS
LIN {X -34.0832,Y -120.5913,Z 143,A -108.7101,B 22.5624,C -0.9577,E1 22.5374,E2 555.8258} C_DIS
LIN {X -38.4218,Y -119.2798,Z 143,A -110.7375,B 22.5624,C -0.9611,E1 22.532,E2 557.8481} C_DIS
LIN {X -41.1362,Y -118.3707,Z 143,A -112.0658,B 22.5623,C -0.9614,E1 22.5285,E2 559.1785} C_DIS
LIN {X -44.8641,Y -117.01,Z 143,A -113.9294,B 22.5623,C -0.961,E1 22.5236,E2 561.0475} C_DIS
LIN {X -48.7838,Y -115.4305,Z 143,A -115.765,B 22.5621,C -0.9671,E1 22.5188,E2 562.8719} C_DIS
LIN {X -51.0749,Y -114.434,Z 143,A -116.9881,B 22.5621,C -0.9649,E1 22.5157,E2 564.1038} C_DIS
LIN {X -54.5084,Y -112.8402,Z 143,A -118.6529,B 22.562,C -0.9697,E1 22.5115,E2 565.7608} C_DIS
LIN {X -57.3411,Y -111.4274,Z 143,A -120.2674,B 22.5622,C -0.9645,E1 22.5075,E2 567.3938} C_DIS
LIN {X -61.0412,Y -109.4457,Z 143,A -122.1925,B 22.5621,C -0.9669,E1 22.5027,E2 569.319} C_DIS
LIN {X -65.5906,Y -106.7807,Z 143,A -124.5579,B 22.5619,C -0.9723,E1 22.4971,E2 571.6782} C_DIS
LIN {X -69.1834,Y -104.4892,Z 143,A -126.555,B 22.5619,C -0.9733,E1 22.4924,E2 573.6799} C_DIS
LIN {X -73.8446,Y -101.249,Z 143,A -129.155,B 22.5616,C -0.9775,E1 22.4865,E2 576.279} C_DIS
LIN {X -77.1234,Y -98.7743,Z 143,A -131.0287,B 22.5615,C -0.9811,E1 22.4823,E2 578.151} C_DIS
LIN {X -81.037,Y -95.5891,Z 143,A -133.063,B 22.5608,C -0.9967,E1 22.478,E2 580.153} C_DIS
LIN {X -83.0142,Y -93.8769,Z 143,A -134.5399,B 22.5612,C -0.9874,E1 22.4748,E2 581.6608} C_DIS
LIN {X -86.2917,Y -90.8743,Z 143,A -136.6192,B 22.5612,C -0.9896,E1 22.4706,E2 583.7438} C_DIS
LIN {X -89.302,Y -87.9173,Z 143,A -138.4713,B 22.5608,C -0.9969,E1 22.4669,E2 585.5857} C_DIS
LIN {X -92.0702,Y -85.0141,Z 143,A -140.3253,B 22.5608,C -1.0001,E1 22.4634,E2 587.4404} C_DIS
LIN {X -94.7354,Y -82.0338,Z 143,A -142.2329,B 22.5607,C -1.001,E1 22.4599,E2 589.3553} C_DIS
LIN {X -97.5576,Y -78.6559,Z 143,A -144.2951,B 22.5606,C -1.0037,E1 22.4562,E2 591.421} C_DIS
LIN {X -100.3546,Y -75.0551,Z 143,A -146.3239,B 22.5602,C -1.011,E1 22.4528,E2 593.4414} C_DIS
LIN {X -102.6796,Y -71.8418,Z 143,A -148.1608,B 22.5601,C -1.0146,E1 22.4498,E2 595.2791} C_DIS
LIN {X -105.2324,Y -68.0474,Z 143,A -150.1802,B 22.5597,C -1.0229,E1 22.4467,E2 597.2882} C_DIS
LIN {X -107.3944,Y -64.5816,Z 143,A -152.1546,B 22.5597,C -1.0235,E1 22.4438,E2 599.2724} C_DIS
LIN {X -109.6114,Y -60.742,Z 143,A -154.1548,B 22.5594,C -1.03,E1 22.4411,E2 601.2672} C_DIS
LIN {X -111.1274,Y -57.919,Z 143,A -155.5019,B 22.559,C -1.0388,E1 22.4393,E2 602.5992} C_DIS
LIN {X -113.3021,Y -53.5415,Z 143,A -157.722,B 22.5587,C -1.0456,E1 22.4366,E2 604.8149} C_DIS
LIN {X -114.5151,Y -50.8936,Z 143,A -159.0812,B 22.5587,C -1.0483,E1 22.435,E2 606.1754} C_DIS
LIN {X -115.6561,Y -48.2436,Z 143,A -160.4644,B 22.5586,C -1.0495,E1 22.4335,E2 607.5641} C_DIS
LIN {X -116.9032,Y -45.1388,Z 143,A -162.0248,B 22.5584,C -1.0527,E1 22.4319,E2 609.1258} C_DIS
LIN {X -117.9999,Y -42.1892,Z 143,A -163.4479,B 22.5582,C -1.0576,E1 22.4306,E2 610.5451} C_DIS
LIN {X -119.2702,Y -38.4519,Z 143,A -165.8089,B 22.559,C -1.0408,E1 22.4285,E2 612.9652} C_DIS
LIN {X -120.5182,Y -34.3448,Z 143,A -167.1651,B 22.5576,C -1.0708,E1 22.4275,E2 614.2516} C_DIS
LIN {X -121.617,Y -30.2243,Z 143,A -169.1948,B 22.5575,C -1.0736,E1 22.426,E2 616.2873} C_DIS
LIN {X -122.7753,Y -25.1014,Z 143,A -171.7106,B 22.5574,C -1.0765,E1 22.4245,E2 618.8121} C_DIS
LIN {X -123.6384,Y -20.431,Z 143,A -173.6757,B 22.5567,C -1.0915,E1 22.4236,E2 620.7509} C_DIS
LIN {X -124.04,Y -17.8311,Z 143,A -175.051,B 22.5568,C -1.0884,E1 22.423,E2 622.1435} C_DIS
LIN {X -124.5331,Y -13.9904,Z 143,A -176.9268,B 22.5568,C -1.0898,E1 22.4224,E2 624.0283} C_DIS
LIN {X -124.8955,Y -10.2509,Z 143,A -178.6637,B 22.5565,C -1.0945,E1 22.4219,E2 625.7645} C_DIS
LIN {X -125.1599,Y -6.2375,Z 143,A 179.5783,B 22.5561,C -1.1036,E1 22.4216,E2 627.5106} C_DIS
LIN {X -125.2956,Y -2.2209,Z 143,A 177.7502,B 22.5558,C -1.1098,E1 22.4216,E2 629.3347} C_DIS
LIN {X -125.3088,Y 1.4258,Z 143,A 175.9383,B 22.5558,C -1.1094,E1 22.4216,E2 631.1599} C_DIS
LIN {X -125.2078,Y 5.1955,Z 143,A 174.347,B 22.5554,C -1.1202,E1 22.4216,E2 632.7336} C_DIS
LIN {X -124.99,Y 9.0219,Z 143,A 172.5463,B 22.5552,C -1.1239,E1 22.422,E2 634.5366} C_DIS
LIN {X -124.6513,Y 12.8913,Z 143,A 170.6606,B 22.5552,C -1.1253,E1 22.4225,E2 636.4316} C_DIS
LIN {X -123.8949,Y 18.8162,Z 143,A 167.9517,B 22.5547,C -1.1349,E1 22.4235,E2 639.1334} C_DIS
LIN {X -123.2981,Y 22.3947,Z 143,A 166.2156,B 22.5545,C -1.1371,E1 22.4243,E2 640.8752} C_DIS
LIN {X -122.6245,Y 25.8352,Z 143,A 164.6254,B 22.5543,C -1.1427,E1 22.4252,E2 642.4612} C_DIS
LIN {X -121.6708,Y 30.0081,Z 143,A 162.8095,B 22.5537,C -1.1545,E1 22.4264,E2 644.2582} C_DIS
LIN {X -120.8499,Y 33.1585,Z 143,A 161.1573,B 22.5538,C -1.1527,E1 22.4276,E2 645.9259} C_DIS
LIN {X -119.8455,Y 36.618,Z 143,A 159.4547,B 22.5537,C -1.1556,E1 22.429,E2 647.6318} C_DIS
LIN {X -118.7006,Y 40.1789,Z 143,A 157.7429,B 22.5534,C -1.1608,E1 22.4305,E2 649.3409} C_DIS
LIN {X -117.421,Y 43.7737,Z 143,A 156.0015,B 22.5531,C -1.1663,E1 22.4321,E2 651.0789} C_DIS
LIN {X -116.0616,Y 47.2618,Z 143,A 154.4063,B 22.5527,C -1.1762,E1 22.4338,E2 652.6583} C_DIS
LIN {X -113.6438,Y 52.8101,Z 143,A 151.5789,B 22.5524,C -1.1821,E1 22.437,E2 655.4876} C_DIS
LIN {X -111.8008,Y 56.6076,Z 143,A 149.5884,B 22.5522,C -1.1854,E1 22.4394,E2 657.4816} C_DIS
LIN {X -108.7566,Y 62.2598,Z 143,A 147.0378,B 22.551,C -1.2092,E1 22.4428,E2 659.9848} C_DIS
LIN {X -106.3103,Y 66.3506,Z 143,A 144.4327,B 22.5515,C -1.1983,E1 22.4466,E2 662.6334} C_DIS
LIN {X -103.9743,Y 69.955,Z 143,A 142.486,B 22.5512,C -1.2045,E1 22.4496,E2 664.575} C_DIS
LIN {X -101.6572,Y 73.2814,Z 143,A 140.5543,B 22.5512,C -1.2064,E1 22.4527,E2 666.5123} C_DIS
LIN {X -99.3286,Y 76.4081,Z 143,A 138.6535,B 22.5512,C -1.2064,E1 22.4559,E2 668.4232} C_DIS
LIN {X -96.235,Y 80.2695,Z 143,A 136.5778,B 22.5505,C -1.2197,E1 22.4596,E2 670.4748} C_DIS
LIN {X -93.9359,Y 82.9475,Z 143,A 134.9445,B 22.5503,C -1.223,E1 22.4625,E2 672.1077} C_DIS
LIN {X -91.356,Y 85.781,Z 143,A 133.2289,B 22.55,C -1.2288,E1 22.4658,E2 673.8166} C_DIS
LIN {X -88.6755,Y 88.5494,Z 143,A 131.4209,B 22.5499,C -1.2312,E1 22.4693,E2 675.627} C_DIS
LIN {X -86.1413,Y 91.0162,Z 143,A 129.8032,B 22.5497,C -1.235,E1 22.4726,E2 677.2424} C_DIS
LIN {X -83.4515,Y 93.4887,Z 143,A 127.8594,B 22.55,C -1.2278,E1 22.4767,E2 679.2138} C_DIS
LIN {X -79.6426,Y 96.7545,Z 143,A 125.7154,B 22.5495,C -1.2388,E1 22.4812,E2 681.338} C_DIS
LIN {X -76.3934,Y 99.3398,Z 143,A 123.7977,B 22.5493,C -1.2421,E1 22.4854,E2 683.2552} C_DIS
LIN {X -72.9375,Y 101.9037,Z 143,A 121.8886,B 22.549,C -1.2484,E1 22.4897,E2 685.1551} C_DIS
LIN {X -69.341,Y 104.3846,Z 143,A 119.9701,B 22.5486,C -1.2555,E1 22.4941,E2 687.0623} C_DIS
LIN {X -66.7095,Y 106.0855,Z 143,A 118.1165,B 22.5494,C -1.2411,E1 22.4986,E2 688.9603} C_DIS
LIN {X -63.6707,Y 107.9367,Z 143,A 116.4221,B 22.5494,C -1.2412,E1 22.5027,E2 690.6601} C_DIS
LIN {X -60.3203,Y 109.8443,Z 143,A 115.0264,B 22.5484,C -1.2592,E1 22.506,E2 692.0133} C_DIS
LIN {X -57.0195,Y 111.5911,Z 143,A 113.2617,B 22.5484,C -1.2597,E1 22.5104,E2 693.7822} C_DIS
LIN {X -53.0966,Y 113.5114,Z 143,A 111.251,B 22.5482,C -1.2621,E1 22.5154,E2 695.7922} C_DIS
LIN {X -49.0794,Y 115.3061,Z 143,A 109.3911,B 22.5478,C -1.2713,E1 22.5201,E2 697.633} C_DIS
LIN {X -45.6987,Y 116.6855,Z 143,A 107.6077,B 22.5478,C -1.2689,E1 22.5248,E2 699.4272} C_DIS
LIN {X -42.0654,Y 118.0445,Z 143,A 104.9346,B 22.5497,C -1.2341,E1 22.5321,E2 702.1971} C_DIS
LIN {X -35.9286,Y 120.0562,Z 143,A 102.814,B 22.5477,C -1.2716,E1 22.5375,E2 704.2238} C_DIS
LIN {X -29.3203,Y 121.8366,Z 143,A 99.8349,B 22.5472,C -1.2809,E1 22.5455,E2 707.1834} C_DIS
LIN {X -25.8188,Y 122.628,Z 143,A 98.2186,B 22.5472,C -1.2834,E1 22.5499,E2 708.7957} C_DIS
LIN {X -23.395,Y 123.1119,Z 143,A 97.0055,B 22.5472,C -1.2808,E1 22.5532,E2 710.017} C_DIS
LIN {X -19.2883,Y 123.8218,Z 143,A 95.1087,B 22.5472,C -1.2825,E1 22.5585,E2 711.9115} C_DIS
LIN {X -15.6182,Y 124.3398,Z 143,A 93.28,B 22.5474,C -1.2778,E1 22.5636,E2 713.7538} C_DIS
LIN {X -11.1825,Y 124.8168,Z 143,A 91.1171,B 22.5476,C -1.2736,E1 22.5696,E2 715.929} C_DIS
LIN {X -6.1899,Y 125.1622,Z 143,A 89.1686,B 22.5468,C -1.2888,E1 22.5749,E2 717.8385} C_DIS
LIN {X -3.5133,Y 125.266,Z 143,A 87.8158,B 22.5471,C -1.2837,E1 22.5787,E2 719.2048} C_DIS
LIN {X 0.8076,Y 125.3127,Z 143,A 85.9164,B 22.5469,C -1.2873,E1 22.584,E2 721.0948} C_DIS
LIN {X 4.6701,Y 125.2283,Z 143,A 84.1478,B 22.5469,C -1.2873,E1 22.5889,E2 722.8628} C_DIS
LIN {X 8.3451,Y 125.0386,Z 143,A 82.5042,B 22.5469,C -1.289,E1 22.5935,E2 724.5014} C_DIS
LIN {X 10.8311,Y 124.8465,Z 143,A 81.3534,B 22.5469,C -1.2885,E1 22.5967,E2 725.653} C_DIS
LIN {X 13.7495,Y 124.559,Z 143,A 79.8488,B 22.5472,C -1.2812,E1 22.6009,E2 727.1754} C_DIS
LIN {X 17.8478,Y 124.0376,Z 143,A 77.996,B 22.5472,C -1.2823,E1 22.6061,E2 729.0237} C_DIS
LIN {X 21.8643,Y 123.3931,Z 143,A 76.1985,B 22.5471,C -1.2843,E1 22.611,E2 730.8138} C_DIS
LIN {X 25.3289,Y 122.729,Z 143,A 74.6233,B 22.5471,C -1.2852,E1 22.6153,E2 732.3845} C_DIS
LIN {X 28.8395,Y 121.9524,Z 143,A 72.8997,B 22.5472,C -1.2808,E1 22.62,E2 734.1169} C_DIS
LIN {X 32.256,Y 121.0924,Z 143,A 71.1076,B 22.5477,C -1.2719,E1 22.6249,E2 735.929} C_DIS
LIN {X 36.5248,Y 119.874,Z 143,A 69.3301,B 22.5472,C -1.2814,E1 22.6296,E2 737.6784} C_DIS
LIN {X 39.9459,Y 118.7782,Z 143,A 67.6746,B 22.5473,C -1.2794,E1 22.634,E2 739.3354} C_DIS
LIN {X 42.7871,Y 117.7843,Z 143,A 66.1492,B 22.5477,C -1.2716,E1 22.638,E2 740.8775} C_DIS
LIN {X 46.5062,Y 116.3662,Z 143,A 64.4601,B 22.5475,C -1.2755,E1 22.6424,E2 742.5523} C_DIS
LIN {X 49.9252,Y 114.9404,Z 143,A 62.8178,B 22.5475,C -1.276,E1 22.6466,E2 744.1892} C_DIS
LIN {X 53.3446,Y 113.3961,Z 143,A 60.5678,B 22.5489,C -1.2504,E1 22.6525,E2 746.4993} C_DIS
LIN {X 57.0886,Y 111.5559,Z 143,A 59.1687,B 22.5478,C -1.2703,E1 22.6558,E2 747.8422} C_DIS
LIN {X 61.756,Y 109.044,Z 143,A 56.8081,B 22.5478,C -1.2697,E1 22.6616,E2 750.1967} C_DIS
LIN {X 64.9849,Y 107.1505,Z 143,A 55.0306,B 22.5481,C -1.2642,E1 22.6658,E2 751.9824} C_DIS
LIN {X 68.5829,Y 104.8846,Z 143,A 52.0807,B 22.5506,C -1.2166,E1 22.673,E2 755.0451} C_DIS
LIN {X 74.2048,Y 100.9846,Z 143,A 49.7039,B 22.5492,C -1.2444,E1 22.6782,E2 757.3402} C_DIS
LIN {X 76.8061,Y 99.0205,Z 143,A 48.6612,B 22.5483,C -1.2618,E1 22.6804,E2 758.3336} C_DIS
LIN {X 79.232,Y 97.0903,Z 143,A 47.0571,B 22.5488,C -1.2507,E1 22.6839,E2 759.9596} C_DIS
LIN {X 82.6063,Y 94.2365,Z 143,A 45.0163,B 22.5491,C -1.2458,E1 22.6883,E2 762.0041} C_DIS
LIN {X 85.7904,Y 91.3473,Z 143,A 43.0983,B 22.5492,C -1.244,E1 22.6922,E2 763.9182} C_DIS
LIN {X 88.7142,Y 88.5104,Z 143,A 41.2003,B 22.5495,C -1.2384,E1 22.696,E2 765.8217} C_DIS
LIN {X 91.562,Y 85.561,Z 143,A 39.4001,B 22.5495,C -1.2377,E1 22.6994,E2 767.6151} C_DIS
LIN {X 94.2399,Y 82.6024,Z 143,A 37.5137,B 22.5499,C -1.2307,E1 22.7029,E2 769.5102} C_DIS
LIN {X 99.7368,Y 75.8743,Z 143,A 33.8696,B 22.5496,C -1.2362,E1 22.7093,E2 773.121} C_DIS
LIN {X 102.1864,Y 72.5419,Z 143,A 31.8247,B 22.5502,C -1.2244,E1 22.7127,E2 775.1854} C_DIS
LIN {X 104.3107,Y 69.4518,Z 143,A 30.0601,B 22.5506,C -1.2177,E1 22.7155,E2 776.9575} C_DIS
LIN {X 106.6094,Y 65.8699,Z 143,A 27.5931,B 22.552,C -1.1888,E1 22.7192,E2 779.4856} C_DIS
LIN {X 108.8687,Y 62.0633,Z 143,A 26.2818,B 22.5506,C -1.216,E1 22.7209,E2 780.7187} C_DIS
LIN {X 110.4966,Y 59.1168,Z 143,A 24.3871,B 22.5517,C -1.1954,E1 22.7235,E2 782.6556} C_DIS
LIN {X 112.3224,Y 55.5649,Z 143,A 22.8189,B 22.5513,C -1.2022,E1 22.7254,E2 784.1968} C_DIS
LIN {X 113.7603,Y 52.5581,Z 143,A 21.319,B 22.5515,C -1.199,E1 22.7272,E2 785.6959} C_DIS
LIN {X 115.0489,Y 49.6742,Z 143,A 19.6247,B 22.5523,C -1.1834,E1 22.7291,E2 787.4206} C_DIS
LIN {X 116.5036,Y 46.1655,Z 143,A 18.0801,B 22.5521,C -1.1871,E1 22.7307,E2 788.9457} C_DIS
LIN {X 117.8574,Y 42.5845,Z 143,A 16.3219,B 22.5524,C -1.1816,E1 22.7324,E2 790.7072} C_DIS
LIN {X 118.8914,Y 39.6058,Z 143,A 14.9342,B 22.5524,C -1.1798,E1 22.7337,E2 792.0908} C_DIS
LIN {X 119.8992,Y 36.4422,Z 143,A 13.0469,B 22.5535,C -1.1582,E1 22.7353,E2 794.0222} C_DIS
LIN {X 120.9383,Y 32.8339,Z 143,A 11.8053,B 22.5527,C -1.1749,E1 22.7362,E2 795.2124} C_DIS
LIN {X 121.8112,Y 29.4255,Z 143,A 10.0962,B 22.5532,C -1.1653,E1 22.7373,E2 796.9353} C_DIS
LIN {X 122.5557,Y 26.1538,Z 143,A 8.6527,B 22.5532,C -1.1648,E1 22.7382,E2 798.3708} C_DIS
LIN {X 123.1717,Y 23.082,Z 143,A 7.0859,B 22.5537,C -1.1541,E1 22.739,E2 799.9552} C_DIS
LIN {X 123.8497,Y 19.108,Z 143,A 5.3736,B 22.5537,C -1.1544,E1 22.7398,E2 801.6553} C_DIS
LIN {X 124.403,Y 15.0935,Z 143,A 3.521,B 22.554,C -1.1486,E1 22.7405,E2 803.5108} C_DIS
LIN {X 124.7809,Y 11.5662,Z 143,A 1.8404,B 22.5544,C -1.1407,E1 22.7409,E2 805.2007} C_DIS
LIN {X 125.1239,Y 6.9519,Z 143,A -0.2908,B 22.5547,C -1.1332,E1 22.7413,E2 807.3372} C_DIS
LIN {X 125.2542,Y 3.9368,Z 143,A -1.4594,B 22.5545,C -1.1386,E1 22.7414,E2 808.4839} C_DIS
LIN {X 125.3182,Y 0.2937,Z 143,A -3.351,B 22.5552,C -1.1227,E1 22.7414,E2 810.4041} C_DIS
LIN {X 125.2286,Y -4.6619,Z 143,A -5.4535,B 22.5552,C -1.1231,E1 22.7414,E2 812.4916} C_DIS
LIN {X 125.0522,Y -8.1254,Z 143,A -6.9643,B 22.5552,C -1.1215,E1 22.7411,E2 813.9964} C_DIS
LIN {X 124.8142,Y -11.214,Z 143,A -8.5793,B 22.5559,C -1.1076,E1 22.7407,E2 815.6366} C_DIS
LIN {X 124.3666,Y -15.3993,Z 143,A -10.512,B 22.5562,C -1.1011,E1 22.7401,E2 817.5735} C_DIS
LIN {X 123.8891,Y -18.8536,Z 143,A -11.9704,B 22.5562,C -1.1023,E1 22.7395,E2 819.019} C_DIS
LIN {X 123.3209,Y -22.2673,Z 143,A -13.5593,B 22.5564,C -1.0969,E1 22.7387,E2 820.6114} C_DIS
LIN {X 121.773,Y -29.5841,Z 143,A -16.8534,B 22.5567,C -1.0919,E1 22.7368,E2 823.8971} C_DIS
LIN {X 120.9549,Y -32.7718,Z 143,A -18.6673,B 22.5575,C -1.0727,E1 22.7354,E2 825.7491} C_DIS
LIN {X 119.6994,Y -37.0952,Z 143,A -20.4321,B 22.5572,C -1.0799,E1 22.7341,E2 827.4838} C_DIS
LIN {X 118.1314,Y -41.8244,Z 143,A -22.6309,B 22.5574,C -1.0765,E1 22.7321,E2 829.6775} C_DIS
LIN {X 116.5303,Y -46.0979,Z 143,A -24.8615,B 22.558,C -1.0634,E1 22.7298,E2 831.9283} C_DIS
LIN {X 115.2264,Y -49.2637,Z 143,A -26.3755,B 22.558,C -1.0611,E1 22.7282,E2 833.4389} C_DIS
LIN {X 113.2313,Y -53.6897,Z 143,A -28.3199,B 22.5578,C -1.0672,E1 22.726,E2 835.3555} C_DIS
LIN {X 111.5651,Y -57.0706,Z 143,A -30.233,B 22.5584,C -1.0533,E1 22.7236,E2 837.2934} C_DIS
LIN {X 109.7249,Y -60.5371,Z 143,A -32.1183,B 22.5588,C -1.0438,E1 22.721,E2 839.1922} C_DIS
LIN {X 107.4643,Y -64.4655,Z 143,A -34.1834,B 22.5591,C -1.0381,E1 22.7181,E2 841.26} C_DIS
LIN {X 104.0878,Y -69.7856,Z 143,A -36.7849,B 22.5589,C -1.043,E1 22.7142,E2 843.8342} C_DIS
LIN {X 102.5386,Y -72.0425,Z 143,A -38.227,B 22.5594,C -1.0307,E1 22.7119,E2 845.3003} C_DIS
LIN {X 100.3674,Y -75.0379,Z 143,A -40.1514,B 22.5601,C -1.0154,E1 22.7087,E2 847.2541} C_DIS
LIN {X 96.683,Y -79.7289,Z 143,A -42.8073,B 22.5602,C -1.0115,E1 22.704,E2 849.9062} C_DIS
LIN {X 94.3998,Y -82.4192,Z 143,A -44.2524,B 22.5601,C -1.0151,E1 22.7014,E2 851.3347} C_DIS
LIN {X 89.3967,Y -87.8207,Z 143,A -47.3804,B 22.56,C -1.0177,E1 22.6955,E2 854.4405} C_DIS
LIN {X 85.6594,Y -91.4703,Z 143,A -49.9999,B 22.5606,C -1.0014,E1 22.6901,E2 857.0903} C_DIS
LIN {X 80.9881,Y -95.6307,Z 143,A -52.8316,B 22.5609,C -0.9962,E1 22.6842,E2 859.9229} C_DIS
LIN {X 78.5092,Y -97.6759,Z 143,A -54.2805,B 22.5609,C -0.9939,E1 22.681,E2 861.3716} C_DIS
LIN {X 75.1341,Y -100.2958,Z 143,A -56.2603,B 22.5612,C -0.9885,E1 22.6766,E2 863.3572} C_DIS
LIN {X 71.4346,Y -102.963,Z 143,A -58.2956,B 22.5612,C -0.9866,E1 22.672,E2 865.3896} C_DIS
LIN {X 68.3962,Y -105.0059,Z 143,A -59.9781,B 22.5614,C -0.9829,E1 22.6681,E2 867.0753} C_DIS
LIN {X 64.6205,Y -107.3709,Z 143,A -61.891,B 22.5614,C -0.9848,E1 22.6636,E2 868.9767} C_DIS
LIN {X 61.4715,Y -109.204,Z 143,A -63.5932,B 22.5615,C -0.9802,E1 22.6594,E2 870.6851} C_DIS
LIN {X 57.4346,Y -111.3798,Z 143,A -65.5774,B 22.5615,C -0.9817,E1 22.6546,E2 872.659} C_DIS
LIN {X 53.0981,Y -113.5106,Z 143,A -68.1396,B 22.5623,C -0.9623,E1 22.648,E2 875.2641} C_DIS
LIN {X 47.9065,Y -115.7969,Z 143,A -70.4651,B 22.5619,C -0.9706,E1 22.6421,E2 877.5618} C_DIS
LIN {X 44.2455,Y -117.2443,Z 143,A -73.0979,B 22.5635,C -0.931,E1 22.635,E2 880.2912} C_DIS
LIN {X 38.6475,Y -119.2077,Z 143,A -75.6759,B 22.5635,C -0.9337,E1 22.6282,E2 882.8568} C_DIS
LIN {X 33.6424,Y -120.7146,Z 143,A -77.2781,B 22.5621,C -0.9661,E1 22.6241,E2 884.3717} C_DIS
LIN {X 30.4713,Y -121.5543,Z 143,A -78.9205,B 22.5624,C -0.9582,E1 22.6196,E2 886.0318} C_DIS
LIN {X 26.4123,Y -122.4999,Z 143,A -80.7864,B 22.5624,C -0.9582,E1 22.6145,E2 887.8947} C_DIS
LIN {X 22.9342,Y -123.2,Z 143,A -82.297,B 22.5623,C -0.9618,E1 22.6104,E2 889.394} C_DIS
LIN {X 20.5103,Y -123.6252,Z 143,A -83.4804,B 22.5624,C -0.9584,E1 22.6071,E2 890.5848} C_DIS
LIN {X 16.2449,Y -124.2577,Z 143,A -85.5119,B 22.5626,C -0.9545,E1 22.6015,E2 892.6247} C_DIS
LIN {X 12.8798,Y -124.6526,Z 143,A -87.0921,B 22.5626,C -0.9522,E1 22.5971,E2 894.2095} C_DIS
LIN {X 8.4453,Y -125.0321,Z 143,A -89.0387,B 22.5626,C -0.9552,E1 22.5917,E2 896.1474} C_DIS
LIN {X 4.598,Y -125.2311,Z 143,A -90.6697,B 22.5623,C -0.9603,E1 22.5872,E2 897.7644} C_DIS
LIN {X 1.4493,Y -125.3083,Z 143,A -92.333,B 22.5628,C -0.9501,E1 22.5825,E2 899.454} C_DIS
LIN {X 1.4493,Y -125.3083,Z 143,A -92.333,B 22.5628,C -0.9501,E1 22.5825,E2 899.454} C_DIS
Enddeposition()
LIN {X 0.8945,Y -124.3442,Z 143,A -91.8125,B 21.6348,C -0.8364,E1 21.6519,E2 899.1225} C_DIS
Startdeposition()
$VEL.CP = VEL_PRINT
LIN {X 3.0426,Y -124.3129,Z 143,A -90.4758,B 21.6342,C -0.8512,E1 21.6557,E2 897.7458} C_DIS
LIN {X 6.0881,Y -124.2004,Z 143,A -89.0915,B 21.6342,C -0.8509,E1 21.6596,E2 896.3629} C_DIS
LIN {X 9.1487,Y -124.0124,Z 143,A -87.7032,B 21.6342,C -0.8504,E1 21.6634,E2 894.9767} C_DIS
LIN {X 12.1856,Y -123.7512,Z 143,A -86.3375,B 21.6343,C -0.8495,E1 21.6672,E2 893.6145} C_DIS
LIN {X 15.2143,Y -123.416,Z 143,A -84.9385,B 21.6343,C -0.8501,E1 21.6711,E2 892.2151} C_DIS
LIN {X 18.4919,Y -122.9678,Z 143,A -83.3159,B 21.6341,C -0.8553,E1 21.6756,E2 890.5801} C_DIS
LIN {X 21.2597,Y -122.5201,Z 143,A -82.0287,B 21.6341,C -0.856,E1 21.6792,E2 889.2925} C_DIS
LIN {X 24.2583,Y -121.9613,Z 143,A -80.6347,B 21.6341,C -0.8566,E1 21.683,E2 887.8987} C_DIS
LIN {X 27.4785,Y -121.2753,Z 143,A -79.2707,B 21.6342,C -0.8514,E1 21.6866,E2 886.5509} C_DIS
LIN {X 30.2066,Y -120.6251,Z 143,A -77.8394,B 21.634,C -0.8586,E1 21.6906,E2 885.1026} C_DIS
LIN {X 33.1948,Y -119.837,Z 143,A -76.49,B 21.634,C -0.8569,E1 21.6942,E2 883.7604} C_DIS
LIN {X 36.1078,Y -118.9916,Z 143,A -75.0962,B 21.634,C -0.8583,E1 21.6979,E2 882.3657} C_DIS
LIN {X 39.0025,Y -118.0745,Z 143,A -73.7019,B 21.634,C -0.8597,E1 21.7016,E2 880.9706} C_DIS
LIN {X 42.0994,Y -117.0057,Z 143,A -72.1117,B 21.6337,C -0.8651,E1 21.7058,E2 879.3696} C_DIS
LIN {X 44.9812,Y -115.9283,Z 143,A -70.7929,B 21.6338,C -0.8627,E1 21.7093,E2 878.0607} C_DIS
LIN {X 47.5812,Y -114.8862,Z 143,A -69.4324,B 21.6336,C -0.8675,E1 21.7128,E2 876.6909} C_DIS
LIN {X 50.8261,Y -113.4873,Z 143,A -67.9313,B 21.6337,C -0.8644,E1 21.7166,E2 875.2025} C_DIS
LIN {X 53.1639,Y -112.4122,Z 143,A -66.6224,B 21.6335,C -0.8716,E1 21.72,E2 873.8781} C_DIS
LIN {X 55.9077,Y -111.0734,Z 143,A -65.2146,B 21.6334,C -0.8739,E1 21.7235,E2 872.4686} C_DIS
LIN {X 58.8441,Y -109.5468,Z 143,A -63.7728,B 21.6334,C -0.8728,E1 21.727,E2 871.0346} C_DIS
LIN {X 61.2965,Y -108.1942,Z 143,A -62.4246,B 21.6332,C -0.8775,E1 21.7303,E2 869.6782} C_DIS
LIN {X 64.14,Y -106.5328,Z 143,A -61.0156,B 21.6333,C -0.8755,E1 21.7337,E2 868.2798} C_DIS
LIN {X 66.7309,Y -104.9297,Z 143,A -59.6091,B 21.6333,C -0.8782,E1 21.737,E2 866.8712} C_DIS
LIN {X 69.079,Y -103.3984,Z 143,A -58.2483,B 21.633,C -0.8838,E1 21.7402,E2 865.5007} C_DIS
LIN {X 71.8886,Y -101.4654,Z 143,A -56.7927,B 21.633,C -0.8818,E1 21.7435,E2 864.0563} C_DIS
LIN {X 74.0757,Y -99.8798,Z 143,A -55.4638,B 21.6328,C -0.8881,E1 21.7465,E2 862.7161} C_DIS
LIN {X 77.0964,Y -97.5674,Z 143,A -53.6049,B 21.6325,C -0.8965,E1 21.7507,E2 860.8426} C_DIS
LIN {X 80.0445,Y -95.1632,Z 143,A -51.8718,B 21.6324,C -0.8994,E1 21.7544,E2 859.1093} C_DIS
LIN {X 82.9447,Y -92.646,Z 143,A -50.0907,B 21.6322,C -0.9039,E1 21.7581,E2 857.3242} C_DIS
LIN {X 86.2823,Y -89.5465,Z 143,A -48.0068,B 21.632,C -0.9082,E1 21.7623,E2 855.239} C_DIS
LIN {X 89.053,Y -86.7919,Z 143,A -46.205,B 21.6319,C -0.9126,E1 21.7659,E2 853.4343} C_DIS
LIN {X 92.1386,Y -83.5081,Z 143,A -44.2795,B 21.6319,C -0.911,E1 21.7695,E2 851.523} C_DIS
LIN {X 94.7247,Y -80.5628,Z 143,A -42.3863,B 21.6316,C -0.9195,E1 21.773,E2 849.6171} C_DIS
LIN {X 97.5314,Y -77.142,Z 143,A -40.321,B 21.6313,C -0.926,E1 21.7766,E2 847.5455} C_DIS
LIN {X 100.0264,Y -73.8779,Z 143,A -38.6092,B 21.6314,C -0.9229,E1 21.7795,E2 845.8516} C_DIS
LIN {X 101.7971,Y -71.4183,Z 143,A -37.2069,B 21.6313,C -0.9269,E1 21.7817,E2 844.4464} C_DIS
LIN {X 103.5209,Y -68.8955,Z 143,A -35.8634,B 21.6313,C -0.9279,E1 21.7838,E2 843.108} C_DIS
LIN {X 105.1919,Y -66.3159,Z 143,A -34.4678,B 21.6311,C -0.931,E1 21.7859,E2 841.7125} C_DIS
LIN {X 106.6596,Y -63.9292,Z 143,A -33.0669,B 21.6308,C -0.9395,E1 21.788,E2 840.2969} C_DIS
LIN {X 108.1955,Y -61.2944,Z 143,A -31.7259,B 21.6308,C -0.9407,E1 21.7898,E2 838.961} C_DIS
LIN {X 109.6642,Y -58.6255,Z 143,A -30.1575,B 21.6302,C -0.9521,E1 21.7919,E2 837.3713} C_DIS
LIN {X 111.3656,Y -55.3215,Z 143,A -28.8081,B 21.6307,C -0.9409,E1 21.7936,E2 836.0608} C_DIS
LIN {X 112.788,Y -52.36,Z 143,A -27.0151,B 21.63,C -0.9579,E1 21.7958,E2 834.2332} C_DIS
LIN {X 114.3928,Y -48.7582,Z 143,A -25.21,B 21.6298,C -0.9628,E1 21.7978,E2 832.4265} C_DIS
LIN {X 116.0172,Y -44.7526,Z 143,A -23.3521,B 21.6298,C -0.9628,E1 21.7997,E2 830.5806} C_DIS
LIN {X 117.1617,Y -41.6665,Z 143,A -21.846,B 21.6296,C -0.967,E1 21.8011,E2 829.0732} C_DIS
LIN {X 118.1514,Y -38.7716,Z 143,A -20.4493,B 21.6294,C -0.9707,E1 21.8024,E2 827.6756} C_DIS
LIN {X 119.0637,Y -35.8723,Z 143,A -19.0607,B 21.6293,C -0.9745,E1 21.8035,E2 826.286} C_DIS
LIN {X 120.0356,Y -32.4708,Z 143,A -17.5705,B 21.6293,C -0.9733,E1 21.8046,E2 824.8091} C_DIS
LIN {X 120.667,Y -30.0416,Z 143,A -16.3133,B 21.629,C -0.9815,E1 21.8055,E2 823.5385} C_DIS
LIN {X 121.2919,Y -27.4059,Z 143,A -15.039,B 21.6288,C -0.9866,E1 21.8063,E2 822.259} C_DIS
LIN {X 121.9614,Y -24.2579,Z 143,A -13.5438,B 21.6285,C -0.9918,E1 21.8071,E2 820.76} C_DIS
LIN {X 122.555,Y -21.0561,Z 143,A -12.1604,B 21.6285,C -0.9913,E1 21.8078,E2 819.3875} C_DIS
LIN {X 123.0393,Y -18.0072,Z 143,A -10.6702,B 21.6282,C -0.9989,E1 21.8084,E2 817.8872} C_DIS
LIN {X 123.4449,Y -14.9719,Z 143,A -9.2776,B 21.6281,C -1.0025,E1 21.8089,E2 816.4944} C_DIS
LIN {X 123.7511,Y -12.1868,Z 143,A -7.9393,B 21.6278,C -1.0088,E1 21.8093,E2 815.1486} C_DIS
LIN {X 124.0124,Y -9.1492,Z 143,A -6.5638,B 21.6276,C -1.0119,E1 21.8096,E2 813.7742} C_DIS
LIN {X 124.1995,Y -6.1062,Z 143,A -5.191,B 21.6276,C -1.015,E1 21.8098,E2 812.4027} C_DIS
LIN {X 124.3206,Y -2.7652,Z 143,A -3.6368,B 21.6273,C -1.0205,E1 21.8099,E2 810.8445} C_DIS
LIN {X 124.3538,Y 0.1273,Z 143,A -2.2123,B 21.6269,C -1.0288,E1 21.8099,E2 809.4076} C_DIS
LIN {X 124.3057,Y 3.303,Z 143,A -0.9075,B 21.627,C -1.0264,E1 21.8099,E2 808.1185} C_DIS
LIN {X 124.1694,Y 6.7049,Z 143,A 0.6035,B 21.6269,C -1.0287,E1 21.8097,E2 806.6116} C_DIS
LIN {X 123.9769,Y 9.6348,Z 143,A 1.9634,B 21.6267,C -1.0333,E1 21.8094,E2 805.2488} C_DIS
LIN {X 123.7508,Y 12.1901,Z 143,A 3.1547,B 21.6265,C -1.0375,E1 21.8091,E2 804.0546} C_DIS
LIN {X 123.4153,Y 15.2204,Z 143,A 4.6958,B 21.626,C -1.048,E1 21.8086,E2 802.4958} C_DIS
LIN {X 122.8937,Y 18.9708,Z 143,A 6.3229,B 21.626,C -1.0482,E1 21.8079,E2 800.8795} C_DIS
LIN {X 122.2494,Y 22.7634,Z 143,A 8.2202,B 21.6255,C -1.0593,E1 21.807,E2 798.9654} C_DIS
LIN {X 121.6021,Y 25.9946,Z 143,A 9.5582,B 21.6256,C -1.0558,E1 21.8062,E2 797.6457} C_DIS
LIN {X 120.9856,Y 28.7292,Z 143,A 10.8414,B 21.6255,C -1.0594,E1 21.8054,E2 796.3616} C_DIS
LIN {X 120.1787,Y 31.9341,Z 143,A 12.288,B 21.6255,C -1.0606,E1 21.8044,E2 794.9215} C_DIS
LIN {X 119.4247,Y 34.6485,Z 143,A 13.6384,B 21.6251,C -1.0669,E1 21.8034,E2 793.5634} C_DIS
LIN {X 118.5403,Y 37.5628,Z 143,A 15.031,B 21.625,C -1.0706,E1 21.8022,E2 792.1701} C_DIS
LIN {X 117.5845,Y 40.4555,Z 143,A 16.4848,B 21.6247,C -1.077,E1 21.8009,E2 790.7087} C_DIS
LIN {X 116.472,Y 43.5541,Z 143,A 17.9304,B 21.6246,C -1.0782,E1 21.7995,E2 789.2692} C_DIS
LIN {X 115.4617,Y 46.1669,Z 143,A 19.2101,B 21.6244,C -1.0815,E1 21.7982,E2 787.989} C_DIS
LIN {X 114.1272,Y 49.3726,Z 143,A 20.7897,B 21.6243,C -1.0851,E1 21.7965,E2 786.4097} C_DIS
LIN {X 112.9511,Y 52.0071,Z 143,A 22.2347,B 21.6238,C -1.094,E1 21.7948,E2 784.9499} C_DIS
LIN {X 111.0741,Y 55.9064,Z 143,A 24.1785,B 21.6237,C -1.0973,E1 21.7924,E2 783.0095} C_DIS
LIN {X 109.4588,Y 59.0079,Z 143,A 25.6662,B 21.6237,C -1.0962,E1 21.7905,E2 781.534} C_DIS
LIN {X 108.201,Y 61.2847,Z 143,A 26.9548,B 21.6234,C -1.1034,E1 21.7887,E2 780.2338} C_DIS
LIN {X 106.5472,Y 64.1162,Z 143,A 28.5439,B 21.623,C -1.1109,E1 21.7864,E2 778.6341} C_DIS
LIN {X 104.2337,Y 67.812,Z 143,A 30.3928,B 21.6231,C -1.109,E1 21.7837,E2 776.8011} C_DIS
LIN {X 102.4014,Y 70.5487,Z 143,A 31.8557,B 21.6231,C -1.1105,E1 21.7814,E2 775.3429} C_DIS
LIN {X 100.7731,Y 72.8556,Z 143,A 33.3231,B 21.6225,C -1.121,E1 21.779,E2 773.8553} C_DIS
LIN {X 98.0406,Y 76.4939,Z 143,A 35.4394,B 21.6222,C -1.127,E1 21.7754,E2 771.7348} C_DIS
LIN {X 95.179,Y 80.0256,Z 143,A 37.4767,B 21.6222,C -1.1294,E1 21.7718,E2 769.7021} C_DIS
LIN {X 92.6491,Y 82.9414,Z 143,A 39.2555,B 21.6219,C -1.1334,E1 21.7685,E2 767.9217} C_DIS
LIN {X 89.6159,Y 86.2106,Z 143,A 41.3363,B 21.6216,C -1.139,E1 21.7645,E2 765.8363} C_DIS
LIN {X 86.757,Y 89.0869,Z 143,A 43.1916,B 21.6215,C -1.1424,E1 21.7608,E2 763.9811} C_DIS
LIN {X 83.4233,Y 92.2155,Z 143,A 45.2453,B 21.6214,C -1.1444,E1 21.7566,E2 761.9318} C_DIS
LIN {X 80.195,Y 95.0368,Z 143,A 47.1677,B 21.6213,C -1.1459,E1 21.7525,E2 760.0142} C_DIS
LIN {X 77.1059,Y 97.56,Z 143,A 49.0869,B 21.6209,C -1.1529,E1 21.7483,E2 758.0846} C_DIS
LIN {X 73.6951,Y 100.1607,Z 143,A 50.8465,B 21.6212,C -1.147,E1 21.7444,E2 756.3484} C_DIS
LIN {X 71.6162,Y 101.6575,Z 143,A 52.1083,B 21.6209,C -1.1525,E1 21.7415,E2 755.0768} C_DIS
LIN {X 68.9241,Y 103.5017,Z 143,A 53.6976,B 21.6206,C -1.1587,E1 21.7378,E2 753.4771} C_DIS
LIN {X 65.956,Y 105.4183,Z 143,A 55.3136,B 21.6206,C -1.1607,E1 21.734,E2 751.8618} C_DIS
LIN {X 62.4092,Y 107.5557,Z 143,A 57.0178,B 21.6208,C -1.1548,E1 21.73,E2 750.1797} C_DIS
LIN {X 59.6651,Y 109.1019,Z 143,A 58.4554,B 21.6208,C -1.1562,E1 21.7265,E2 748.7432} C_DIS
LIN {X 57.0563,Y 110.4886,Z 143,A 59.8733,B 21.6205,C -1.1604,E1 21.7229,E2 747.3185} C_DIS
LIN {X 54.3433,Y 111.8482,Z 143,A 61.3964,B 21.6202,C -1.1675,E1 21.7191,E2 745.7811} C_DIS
LIN {X 51.7829,Y 113.0548,Z 143,A 62.589,B 21.6203,C -1.1643,E1 21.7161,E2 744.6006} C_DIS
LIN {X 48.77,Y 114.3877,Z 143,A 64.103,B 21.6203,C -1.1658,E1 21.7122,E2 743.0868} C_DIS
LIN {X 46.1776,Y 115.4574,Z 143,A 65.3891,B 21.6203,C -1.167,E1 21.7089,E2 741.8012} C_DIS
LIN {X 43.1717,Y 116.6152,Z 143,A 66.876,B 21.6201,C -1.1685,E1 21.705,E2 740.314} C_DIS
LIN {X 39.8988,Y 117.776,Z 143,A 68.417,B 21.6201,C -1.1674,E1 21.701,E2 738.7795} C_DIS
LIN {X 37.3297,Y 118.6148,Z 143,A 69.7065,B 21.6201,C -1.1703,E1 21.6975,E2 737.485} C_DIS
LIN {X 34.4162,Y 119.4928,Z 143,A 71.0886,B 21.6201,C -1.1705,E1 21.6938,E2 736.1051} C_DIS
LIN {X 31.286,Y 120.3512,Z 143,A 72.7225,B 21.6197,C -1.1773,E1 21.6894,E2 734.4559} C_DIS
LIN {X 27.2429,Y 121.3291,Z 143,A 74.5275,B 21.6199,C -1.1737,E1 21.6845,E2 732.6636} C_DIS
LIN {X 23.4113,Y 122.1255,Z 143,A 76.1002,B 21.6203,C -1.165,E1 21.6803,E2 731.1169} C_DIS
LIN {X 21.2621,Y 122.5197,Z 143,A 77.4781,B 21.6195,C -1.1808,E1 21.6764,E2 729.6978} C_DIS
LIN {X 18.0087,Y 123.039,Z 143,A 78.8464,B 21.6198,C -1.175,E1 21.6726,E2 728.3467} C_DIS
LIN {X 14.7001,Y 123.4774,Z 143,A 80.3139,B 21.6199,C -1.1725,E1 21.6686,E2 726.8874} C_DIS
LIN {X 12.1884,Y 123.751,Z 143,A 81.6007,B 21.6197,C -1.1777,E1 21.665,E2 725.5874} C_DIS
LIN {X 9.1491,Y 124.0124,Z 143,A 82.9877,B 21.6197,C -1.1771,E1 21.6611,E2 724.2029} C_DIS
LIN {X 6.1072,Y 124.1994,Z 143,A 84.3718,B 21.6197,C -1.1763,E1 21.6573,E2 722.8216} C_DIS
LIN {X 3.0549,Y 124.3126,Z 143,A 85.7869,B 21.6197,C -1.1765,E1 21.6533,E2 721.4064} C_DIS
LIN {X -0.0012,Y 124.3514,Z 143,A 87.3065,B 21.6195,C -1.1808,E1 21.6491,E2 719.8751} C_DIS
LIN {X -3.0487,Y 124.3127,Z 143,A 88.6411,B 21.6197,C -1.1777,E1 21.6454,E2 718.5489} C_DIS
LIN {X -6.0952,Y 124.2,Z 143,A 90.0242,B 21.6197,C -1.1764,E1 21.6415,E2 717.1689} C_DIS
LIN {X -9.139,Y 124.0131,Z 143,A 91.4138,B 21.6197,C -1.1752,E1 21.6376,E2 715.7819} C_DIS
LIN {X -12.1889,Y 123.7509,Z 143,A 92.7862,B 21.6199,C -1.173,E1 21.6338,E2 714.4147} C_DIS
LIN {X -15.2191,Y 123.4155,Z 143,A 94.1896,B 21.6199,C -1.1722,E1 21.6299,E2 713.0124} C_DIS
LIN {X -18.4814,Y 122.9694,Z 143,A 95.8236,B 21.6197,C -1.176,E1 21.6254,E2 711.3665} C_DIS
LIN {X -22.0599,Y 122.3769,Z 143,A 97.3064,B 21.6202,C -1.1672,E1 21.6214,E2 709.9059} C_DIS
LIN {X -25.9926,Y 121.6025,Z 143,A 99.2485,B 21.6201,C -1.1696,E1 21.616,E2 707.9547} C_DIS
LIN {X -28.7273,Y 120.9861,Z 143,A 100.5512,B 21.6201,C -1.1689,E1 21.6125,E2 706.6518} C_DIS
LIN {X -31.9412,Y 120.1768,Z 143,A 102.1952,B 21.6199,C -1.1722,E1 21.608,E2 704.9961} C_DIS
LIN {X -36.455,Y 118.8854,Z 143,A 104.1425,B 21.6205,C -1.1612,E1 21.6029,E2 703.0748} C_DIS
LIN {X -38.9865,Y 118.0798,Z 143,A 105.4652,B 21.6204,C -1.1638,E1 21.5993,E2 701.7424} C_DIS
LIN {X -42.1206,Y 116.998,Z 143,A 106.9991,B 21.6204,C -1.1622,E1 21.5953,E2 700.2093} C_DIS
LIN {X -44.9842,Y 115.9271,Z 143,A 108.3436,B 21.6207,C -1.1578,E1 21.5918,E2 698.8734} C_DIS
LIN {X -47.5856,Y 114.8843,Z 143,A 109.7725,B 21.6205,C -1.1615,E1 21.5881,E2 697.4306} C_DIS
LIN {X -50.6116,Y 113.5833,Z 143,A 111.2294,B 21.6207,C -1.157,E1 21.5844,E2 695.982} C_DIS
LIN {X -53.1591,Y 112.4144,Z 143,A 112.5974,B 21.6207,C -1.1581,E1 21.5809,E2 694.6071} C_DIS
LIN {X -55.9304,Y 111.0619,Z 143,A 114.0264,B 21.6207,C -1.1562,E1 21.5773,E2 693.1789} C_DIS
LIN {X -58.8221,Y 109.5586,Z 143,A 115.4514,B 21.621,C -1.1507,E1 21.5738,E2 691.7641} C_DIS
LIN {X -61.2257,Y 108.2343,Z 143,A 116.7652,B 21.621,C -1.1505,E1 21.5706,E2 690.4464} C_DIS
LIN {X -63.9083,Y 106.6721,Z 143,A 118.2358,B 21.621,C -1.1496,E1 21.5671,E2 688.9731} C_DIS
LIN {X -67.3589,Y 104.5277,Z 143,A 120.1742,B 21.6211,C -1.1487,E1 21.5625,E2 687.0298} C_DIS
LIN {X -70.5609,Y 102.393,Z 143,A 121.7858,B 21.6216,C -1.139,E1 21.5588,E2 685.4383} C_DIS
LIN {X -72.8478,Y 100.7787,Z 143,A 123.1215,B 21.6216,C -1.1382,E1 21.5558,E2 684.0992} C_DIS
LIN {X -75.3938,Y 98.8885,Z 143,A 124.7172,B 21.6216,C -1.1405,E1 21.5522,E2 682.4906} C_DIS
LIN {X -78.7877,Y 96.2062,Z 143,A 126.6217,B 21.6219,C -1.1328,E1 21.5481,E2 680.5987} C_DIS
LIN {X -81.6976,Y 93.7477,Z 143,A 128.3921,B 21.6221,C -1.1296,E1 21.5443,E2 678.8291} C_DIS
LIN {X -84.6334,Y 91.1062,Z 143,A 130.3456,B 21.6221,C -1.1307,E1 21.5403,E2 676.8633} C_DIS
LIN {X -87.9242,Y 87.9353,Z 143,A 132.4764,B 21.6222,C -1.1267,E1 21.536,E2 674.7329} C_DIS
LIN {X -91.0957,Y 84.6446,Z 143,A 134.4556,B 21.6227,C -1.1167,E1 21.5323,E2 672.7708} C_DIS
LIN {X -93.7394,Y 81.7071,Z 143,A 136.3897,B 21.6227,C -1.1165,E1 21.5287,E2 670.8269} C_DIS
LIN {X -96.6016,Y 78.3028,Z 143,A 138.4767,B 21.6229,C -1.1127,E1 21.5249,E2 668.7389} C_DIS
LIN {X -99.1154,Y 75.0954,Z 143,A 140.2059,B 21.6235,C -1.1021,E1 21.522,E2 667.0291} C_DIS
LIN {X -100.925,Y 72.6458,Z 143,A 141.5976,B 21.6237,C -1.0979,E1 21.5197,E2 665.6408} C_DIS
LIN {X -102.6748,Y 70.1504,Z 143,A 143.043,B 21.6237,C -1.0957,E1 21.5174,E2 664.1931} C_DIS
LIN {X -104.7059,Y 67.0806,Z 143,A 144.8096,B 21.6239,C -1.0938,E1 21.5147,E2 662.4214} C_DIS
LIN {X -106.6596,Y 63.9293,Z 143,A 146.5268,B 21.6241,C -1.0893,E1 21.5122,E2 660.7061} C_DIS
LIN {X -108.2104,Y 61.2682,Z 143,A 147.8995,B 21.6243,C -1.0835,E1 21.5104,E2 659.3408} C_DIS
LIN {X -109.6744,Y 58.6065,Z 143,A 149.3629,B 21.6244,C -1.0819,E1 21.5084,E2 657.8726} C_DIS
LIN {X -111.0737,Y 55.9071,Z 143,A 150.7348,B 21.6247,C -1.0767,E1 21.5067,E2 656.5062} C_DIS
LIN {X -112.4083,Y 53.172,Z 143,A 152.1325,B 21.6249,C -1.0725,E1 21.505,E2 655.1113} C_DIS
LIN {X -113.6756,Y 50.4051,Z 143,A 153.5676,B 21.625,C -1.0696,E1 21.5033,E2 653.6748} C_DIS
LIN {X -114.9802,Y 47.3561,Z 143,A 155.0704,B 21.6253,C -1.064,E1 21.5017,E2 652.1774} C_DIS
LIN {X -116.0171,Y 44.7528,Z 143,A 156.4099,B 21.6253,C -1.062,E1 21.5004,E2 650.8346} C_DIS
LIN {X -117.3019,Y 41.2706,Z 143,A 158.0237,B 21.6258,C -1.0531,E1 21.4988,E2 649.2344} C_DIS
LIN {X -118.1557,Y 38.7586,Z 143,A 159.3348,B 21.6258,C -1.0527,E1 21.4977,E2 647.9155} C_DIS
LIN {X -119.0693,Y 35.8539,Z 143,A 160.7471,B 21.626,C -1.0487,E1 21.4965,E2 646.5045} C_DIS
LIN {X -119.8455,Y 33.1643,Z 143,A 162.0703,B 21.6261,C -1.046,E1 21.4955,E2 645.1797} C_DIS
LIN {X -120.6824,Y 29.981,Z 143,A 163.5621,B 21.6264,C -1.0403,E1 21.4945,E2 643.6932} C_DIS
LIN {X -121.3267,Y 27.2534,Z 143,A 164.8891,B 21.6264,C -1.0376,E1 21.4936,E2 642.3644} C_DIS
LIN {X -121.958,Y 24.2743,Z 143,A 166.3262,B 21.6266,C -1.0345,E1 21.4928,E2 640.9259} C_DIS
LIN {X -122.7593,Y 19.8317,Z 143,A 168.5395,B 21.6267,C -1.033,E1 21.4918,E2 638.7012} C_DIS
LIN {X -123.4446,Y 14.9746,Z 143,A 170.6709,B 21.6272,C -1.0209,E1 21.491,E2 636.5878} C_DIS
LIN {X -123.7508,Y 12.19,Z 143,A 172.0942,B 21.6272,C -1.0219,E1 21.4906,E2 635.1519} C_DIS
LIN {X -124.1005,Y 7.8667,Z 143,A 174.0366,B 21.6276,C -1.0134,E1 21.4902,E2 633.2189} C_DIS
LIN {X -124.2753,Y 4.3247,Z 143,A 175.5938,B 21.6279,C -1.0053,E1 21.49,E2 631.6729} C_DIS
LIN {X -124.3461,Y 1.0849,Z 143,A 176.8584,B 21.6285,C -0.9918,E1 21.49,E2 630.436} C_DIS
LIN {X -124.3372,Y -1.7699,Z 143,A 178.5981,B 21.628,C -1.0038,E1 21.49,E2 628.6513} C_DIS
LIN {X -124.1995,Y -6.1057,Z 143,A -179.4777,B 21.6284,C -0.9946,E1 21.4902,E2 626.7386} C_DIS
LIN {X -124.0124,Y -9.149,Z 143,A -178.0813,B 21.6286,C -0.9899,E1 21.4905,E2 625.3452} C_DIS
LIN {X -123.7511,Y -12.1869,Z 143,A -176.703,B 21.6289,C -0.9844,E1 21.4908,E2 623.9721} C_DIS
LIN {X -123.4156,Y -15.2178,Z 143,A -175.1262,B 21.6288,C -0.9866,E1 21.4914,E2 622.3784} C_DIS
LIN {X -122.9673,Y -18.4953,Z 143,A -173.7203,B 21.6292,C -0.9773,E1 21.4919,E2 620.988} C_DIS
LIN {X -122.516,Y -21.2827,Z 143,A -172.3502,B 21.6292,C -0.9759,E1 21.4926,E2 619.612} C_DIS
LIN {X -121.9628,Y -24.2511,Z 143,A -170.9545,B 21.6294,C -0.9718,E1 21.4933,E2 618.2179} C_DIS
LIN {X -121.2725,Y -27.4907,Z 143,A -169.5648,B 21.6298,C -0.9619,E1 21.4941,E2 616.8456} C_DIS
LIN {X -120.6234,Y -30.2134,Z 143,A -168.1254,B 21.6298,C -0.9637,E1 21.4951,E2 615.3913} C_DIS
LIN {X -119.8472,Y -33.1582,Z 143,A -166.7776,B 21.63,C -0.9574,E1 21.4961,E2 614.0517} C_DIS
LIN {X -118.9993,Y -36.0827,Z 143,A -165.3591,B 21.6302,C -0.9537,E1 21.4972,E2 612.6334} C_DIS
Enddeposition()
END
